LIN {X 0,Y 201.547,Z 410.206,A -85,B 0,C 180,E1 -21878.269,E2 -21878.269} C_VEL
LIN {X 0,Y 203.427,Z 397.935,A -85,B 0,C 180,E1 -21879.946,E2 -21879.946} C_VEL
LIN {X 0,Y 205.038,Z 385.054,A -85,B 0,C 180,E1 -21881.241,E2 -21881.241} C_VEL
LIN {X 0,Y 206.208,Z 372.059,A -85,B 0,C 180,E1 -21882.113,E2 -21882.113} C_VEL
LIN {X 0,Y 207.148,Z 353.067,A -85,B 0,C 180,E1 -21882.84,E2 -21882.84} C_VEL
LIN {X 0,Y 209.063,Z 305.006,A -85,B 0,C 180,E1 -21884.444,E2 -21884.444} C_VEL
LIN {X 0,Y 207.505,Z 298.752,A -85,B 0,C 180,E1 -21884.902,E2 -21884.902} C_VEL
LIN {X 0,Y 201.853,Z 283.207,A -85,B 0,C 180,E1 -21886.329,E2 -21886.329} C_VEL
LIN {X 0,Y 196.318,Z 270.427,A -85,B 0,C 180,E1 -21887.718,E2 -21887.718} C_VEL
LIN {X 0,Y 192.917,Z 263.876,A -85,B 0,C 180,E1 -21888.63,E2 -21888.63} C_VEL
LIN {X 0,Y 192.707,Z 263.031,A -85,B 0,C 180,E1 -21889.108,E2 -21889.108} C_VEL
LIN {X 0,Y 192.636,Z 262.96,A -85,B 0,C 180,E1 -21894.234,E2 -21894.234} C_VEL
LIN {X 0,Y 192.624,Z 262.95,A -85,B 0,C 180,E1 -21898.902,E2 -21898.902} C_VEL
LIN {X 0,Y 192.591,Z 262.991,A -85,B 0,C 180,E1 -21903.186,E2 -21903.186} C_VEL
LIN {X 0,Y 192.616,Z 262.98,A -85,B 0,C 180,E1 -21906.629,E2 -21906.629} C_VEL
LIN {X 0,Y 192.586,Z 262.973,A -85,B 0,C 180,E1 -21911.061,E2 -21911.061} C_VEL
LIN {X 0,Y 192.602,Z 262.994,A -85,B 0,C 180,E1 -21916.123,E2 -21916.123} C_VEL
LIN {X 0,Y 192.589,Z 262.963,A -85,B 0,C 180,E1 -21920.025,E2 -21920.025} C_VEL
LIN {X 0,Y 192.579,Z 262.983,A -85,B 0,C 180,E1 -21924.288,E2 -21924.288} C_VEL
LIN {X 0,Y 192.587,Z 262.975,A -85,B 0,C 180,E1 -21929.289,E2 -21929.289} C_VEL
LIN {X 0,Y 192.646,Z 262.94,A -85,B 0,C 180,E1 -21931.701,E2 -21931.701} C_VEL
LIN {X 0,Y 192.698,Z 262.972,A -85,B 0,C 180,E1 -21936.359,E2 -21936.359} C_VEL
LIN {X 0,Y 192.769,Z 262.951,A -85,B 0,C 180,E1 -21941.422,E2 -21941.422} C_VEL
LIN {X 0,Y 192.757,Z 262.917,A -85,B 0,C 180,E1 -21945.224,E2 -21945.224} C_VEL
LIN {X 0,Y 193.012,Z 262.934,A -85,B 0,C 180,E1 -21949.52,E2 -21949.52} C_VEL
LIN {X 0,Y 192.998,Z 262.931,A -85,B 0,C 180,E1 -21953.738,E2 -21953.738} C_VEL
LIN {X 0,Y 193.26,Z 262.855,A -85,B 0,C 180,E1 -21957.925,E2 -21957.925} C_VEL
LIN {X 0,Y 193.438,Z 262.85,A -85,B 0,C 180,E1 -21960.009,E2 -21960.009} C_VEL
LIN {X 0,Y 192.966,Z 262.949,A -85,B 0,C 180,E1 -21964.186,E2 -21964.186} C_VEL
LIN {X 0,Y 193.027,Z 262.904,A -85,B 0,C 180,E1 -21968.383,E2 -21968.383} C_VEL
LIN {X 0,Y 192.805,Z 262.941,A -85,B 0,C 180,E1 -21972.642,E2 -21972.642} C_VEL
LIN {X 0,Y 192.763,Z 262.97,A -85,B 0,C 180,E1 -21976.967,E2 -21976.967} C_VEL
LIN {X 0,Y 192.623,Z 262.954,A -85,B 0,C 180,E1 -21981.408,E2 -21981.408} C_VEL
LIN {X 0,Y 192.656,Z 262.982,A -85,B 0,C 180,E1 -21984.221,E2 -21984.221} C_VEL
LIN {X 0,Y 192.639,Z 262.965,A -85,B 0,C 180,E1 -21988.887,E2 -21988.887} C_VEL
LIN {X 0,Y 192.607,Z 262.996,A -85,B 0,C 180,E1 -21993.194,E2 -21993.194} C_VEL
LIN {X 0,Y 192.562,Z 262.985,A -85,B 0,C 180,E1 -21998.359,E2 -21998.359} C_VEL
LIN {X 0,Y 192.503,Z 262.965,A -85,B 0,C 180,E1 -22003.101,E2 -22003.101} C_VEL
LIN {X 0,Y 192.499,Z 262.962,A -85,B 0,C 180,E1 -22006.913,E2 -22006.913} C_VEL
LIN {X 0,Y 192.609,Z 263.147,A -85,B 0,C 180,E1 -22011.738,E2 -22011.738} C_VEL
LIN {X 0,Y 193.411,Z 266.363,A -85,B 0,C 180,E1 -22013.384,E2 -22013.384} C_VEL
LIN {X 0,Y 198.115,Z 277.207,A -85,B 0,C 180,E1 -22014.69,E2 -22014.69} C_VEL
LIN {X 0,Y 204.165,Z 292.827,A -85,B 0,C 180,E1 -22016.231,E2 -22016.231} C_VEL
LIN {X 0,Y 206.841,Z 301.139,A -85,B 0,C 180,E1 -22016.932,E2 -22016.932} C_VEL
LIN {X 0,Y 207.153,Z 303.933,A -85,B 0,C 180,E1 -22017.085,E2 -22017.085} C_VEL
LIN {X 0,Y 207.117,Z 309.784,A -85,B 0,C 180,E1 -22017.309,E2 -22017.309} C_VEL
LIN {X 0,Y 206.092,Z 315.639,A -85,B 0,C 180,E1 -22017.398,E2 -22017.398} C_VEL
LIN {X 0,Y 202.165,Z 331.222,A -85,B 0,C 180,E1 -22017.472,E2 -22017.472} C_VEL
LIN {X 0,Y 201.68,Z 335.194,A -85,B 0,C 180,E1 -22017.564,E2 -22017.564} C_VEL
LIN {X 0,Y 199.95,Z 375.022,A -85,B 0,C 180,E1 -22018.994,E2 -22018.994} C_VEL
LIN {X 0,Y 198.708,Z 387.932,A -85,B 0,C 180,E1 -22019.809,E2 -22019.809} C_VEL
LIN {X 0,Y 197.203,Z 399.987,A -85,B 0,C 180,E1 -22020.951,E2 -22020.951} C_VEL
LIN {X 0,Y 195.348,Z 411.355,A -85,B 0,C 180,E1 -22022.407,E2 -22022.407} C_VEL
LIN {X 0,Y 193.289,Z 421.772,A -85,B 0,C 180,E1 -22024.132,E2 -22024.132} C_VEL
LIN {X 0,Y 191.373,Z 431.488,A -85,B 0,C 180,E1 -22026.175,E2 -22026.175} C_VEL
LIN {X 0,Y 189.178,Z 441.365,A -85,B 0,C 180,E1 -22028.765,E2 -22028.765} C_VEL
LIN {X 0,Y 187.317,Z 449.442,A -85,B 0,C 180,E1 -22031.404,E2 -22031.404} C_VEL
LIN {X 0,Y 185.503,Z 457.32,A -85,B 0,C 180,E1 -22034.622,E2 -22034.622} C_VEL
LIN {X 0,Y 184.314,Z 463.61,A -85,B 0,C 180,E1 -22037.895,E2 -22037.895} C_VEL
LIN {X 0,Y 183.529,Z 468.588,A -85,B 0,C 180,E1 -22041.19,E2 -22041.19} C_VEL
LIN {X 0,Y 183.125,Z 472.408,A -85,B 0,C 180,E1 -22044.495,E2 -22044.495} C_VEL
LIN {X 0,Y 183.015,Z 475.181,A -85,B 0,C 180,E1 -22047.8,E2 -22047.8} C_VEL
LIN {X 0,Y 183.092,Z 476.483,A -85,B 0,C 180,E1 -22050.001,E2 -22050.001} C_VEL
LIN {X 0,Y 182.991,Z 477.585,A -85,B 0,C 180,E1 -22052.933,E2 -22052.933} C_VEL
LIN {X 0,Y 183.323,Z 477.96,A -85,B 0,C 180,E1 -22056.605,E2 -22056.605} C_VEL
LIN {X 0,Y 184.27,Z 476.977,A -85,B 0,C 180,E1 -22060.994,E2 -22060.994} C_VEL
LIN {X 0,Y 185.114,Z 475.917,A -85,B 0,C 180,E1 -22063.168,E2 -22063.168} C_VEL
LIN {X 0,Y 186.18,Z 474.422,A -85,B 0,C 180,E1 -22065.322,E2 -22065.322} C_VEL
LIN {X 0,Y 188.237,Z 471.426,A -85,B 0,C 180,E1 -22068.504,E2 -22068.504} C_VEL
LIN {X 0,Y 191.001,Z 467.404,A -85,B 0,C 180,E1 -22071.59,E2 -22071.59} C_VEL
LIN {X 0,Y 194.227,Z 462.258,A -85,B 0,C 180,E1 -22074.591,E2 -22074.591} C_VEL
LIN {X 0,Y 197.75,Z 455.833,A -85,B 0,C 180,E1 -22077.518,E2 -22077.518} C_VEL
LIN {X 0,Y 202.024,Z 447.849,A -85,B 0,C 180,E1 -22080.294,E2 -22080.294} C_VEL
LIN {X 0,Y 205.946,Z 439.728,A -85,B 0,C 180,E1 -22082.513,E2 -22082.513} C_VEL
LIN {X 0,Y 210.3,Z 429.83,A -85,B 0,C 180,E1 -22084.62,E2 -22084.62} C_VEL
LIN {X 0,Y 213.87,Z 420.103,A -85,B 0,C 180,E1 -22086.264,E2 -22086.264} C_VEL
LIN {X 0,Y 217.703,Z 407.824,A -85,B 0,C 180,E1 -22087.834,E2 -22087.834} C_VEL
LIN {X 0,Y 220.715,Z 395.821,A -85,B 0,C 180,E1 -22088.968,E2 -22088.968} C_VEL
LIN {X 0,Y 223.081,Z 382.949,A -85,B 0,C 180,E1 -22089.828,E2 -22089.828} C_VEL
LIN {X 0,Y 224.603,Z 369.194,A -85,B 0,C 180,E1 -22090.426,E2 -22090.426} C_VEL
LIN {X 0,Y 226.979,Z 331.617,A -85,B 0,C 180,E1 -22091.565,E2 -22091.565} C_VEL
LIN {X 0,Y 221.2,Z 318.428,A -85,B 0,C 180,E1 -22093.951,E2 -22093.951} C_VEL
LIN {X 0,Y 215.551,Z 307.564,A -85,B 0,C 180,E1 -22096.435,E2 -22096.435} C_VEL
LIN {X 0,Y 209.904,Z 297.83,A -85,B 0,C 180,E1 -22099.202,E2 -22099.202} C_VEL
LIN {X 0,Y 206.451,Z 292.45,A -85,B 0,C 180,E1 -22101.042,E2 -22101.042} C_VEL
LIN {X 0,Y 203.699,Z 288.268,A -85,B 0,C 180,E1 -22102.617,E2 -22102.617} C_VEL
LIN {X 0,Y 199.882,Z 282.7,A -85,B 0,C 180,E1 -22104.997,E2 -22104.997} C_VEL
LIN {X 0,Y 196.957,Z 278.784,A -85,B 0,C 180,E1 -22107.023,E2 -22107.023} C_VEL
LIN {X 0,Y 195.987,Z 277.356,A -85,B 0,C 180,E1 -22107.763,E2 -22107.763} C_VEL
LIN {X 0,Y 190.543,Z 270.611,A -85,B 0,C 180,E1 -22112.417,E2 -22112.417} C_VEL
LIN {X 0,Y 188.641,Z 268.893,A -85,B 0,C 180,E1 -22114.326,E2 -22114.326} C_VEL
LIN {X 0,Y 186.363,Z 266.371,A -85,B 0,C 180,E1 -22117.105,E2 -22117.105} C_VEL
LIN {X 0,Y 185.613,Z 264.245,A -85,B 0,C 180,E1 -22118.763,E2 -22118.763} C_VEL
LIN {X 0,Y 185.542,Z 263.873,A -85,B 0,C 180,E1 -22120.059,E2 -22120.059} C_VEL
LIN {X 0,Y 185.663,Z 263.859,A -85,B 0,C 180,E1 -22122.363,E2 -22122.363} C_VEL
LIN {X 0,Y 185.726,Z 263.851,A -85,B 0,C 180,E1 -22126.868,E2 -22126.868} C_VEL
LIN {X 0,Y 185.984,Z 263.817,A -85,B 0,C 180,E1 -22131.297,E2 -22131.297} C_VEL
LIN {X 0,Y 186.185,Z 263.778,A -85,B 0,C 180,E1 -22137.827,E2 -22137.827} C_VEL
LIN {X 0,Y 186.399,Z 263.758,A -85,B 0,C 180,E1 -22139.99,E2 -22139.99} C_VEL
LIN {X 0,Y 185.946,Z 264.019,A -85,B 0,C 180,E1 -22144.19,E2 -22144.19} C_VEL
LIN {X 0,Y 186.707,Z 266.344,A -85,B 0,C 180,E1 -22145.525,E2 -22145.525} C_VEL
LIN {X 0,Y 188.785,Z 268.646,A -85,B 0,C 180,E1 -22148.015,E2 -22148.015} C_VEL
LIN {X 0,Y 190.993,Z 269.918,A -85,B 0,C 180,E1 -22150.115,E2 -22150.115} C_VEL
LIN {X 0,Y 192.307,Z 272.671,A -85,B 0,C 180,E1 -22151.452,E2 -22151.452} C_VEL
LIN {X 0,Y 194.404,Z 274.827,A -85,B 0,C 180,E1 -22153.185,E2 -22153.185} C_VEL
LIN {X 0,Y 195.644,Z 275.781,A -85,B 0,C 180,E1 -22154.107,E2 -22154.107} C_VEL
LIN {X 0,Y 197.722,Z 279.021,A -85,B 0,C 180,E1 -22155.699,E2 -22155.699} C_VEL
LIN {X 0,Y 199.843,Z 281.118,A -85,B 0,C 180,E1 -22157.093,E2 -22157.093} C_VEL
LIN {X 0,Y 202.443,Z 284.707,A -85,B 0,C 180,E1 -22158.738,E2 -22158.738} C_VEL
LIN {X 0,Y 204.939,Z 288.002,A -85,B 0,C 180,E1 -22160.192,E2 -22160.192} C_VEL
LIN {X 0,Y 208.483,Z 293.32,A -85,B 0,C 180,E1 -22162.146,E2 -22162.146} C_VEL
LIN {X 0,Y 211.835,Z 298.487,A -85,B 0,C 180,E1 -22163.854,E2 -22163.854} C_VEL
LIN {X 0,Y 218.039,Z 309.192,A -85,B 0,C 180,E1 -22166.762,E2 -22166.762} C_VEL
LIN {X 0,Y 223.429,Z 319.688,A -85,B 0,C 180,E1 -22169.04,E2 -22169.04} C_VEL
LIN {X 0,Y 227.273,Z 328.108,A -85,B 0,C 180,E1 -22170.584,E2 -22170.584} C_VEL
LIN {X 0,Y 224.341,Z 370.593,A -85,B 0,C 180,E1 -22171.882,E2 -22171.882} C_VEL
LIN {X 0,Y 222.438,Z 383.985,A -85,B 0,C 180,E1 -22172.584,E2 -22172.584} C_VEL
LIN {X 0,Y 220.078,Z 395.902,A -85,B 0,C 180,E1 -22173.532,E2 -22173.532} C_VEL
LIN {X 0,Y 217.013,Z 407.276,A -85,B 0,C 180,E1 -22174.737,E2 -22174.737} C_VEL
LIN {X 0,Y 213.334,Z 418.666,A -85,B 0,C 180,E1 -22176.357,E2 -22176.357} C_VEL
LIN {X 0,Y 209.3,Z 429.173,A -85,B 0,C 180,E1 -22178.288,E2 -22178.288} C_VEL
LIN {X 0,Y 205.394,Z 438.08,A -85,B 0,C 180,E1 -22180.393,E2 -22180.393} C_VEL
LIN {X 0,Y 201.244,Z 446.261,A -85,B 0,C 180,E1 -22182.829,E2 -22182.829} C_VEL
LIN {X 0,Y 197.654,Z 452.831,A -85,B 0,C 180,E1 -22185.312,E2 -22185.312} C_VEL
LIN {X 0,Y 194.299,Z 458.472,A -85,B 0,C 180,E1 -22187.997,E2 -22187.997} C_VEL
LIN {X 0,Y 190.893,Z 463.723,A -85,B 0,C 180,E1 -22191.253,E2 -22191.253} C_VEL
LIN {X 0,Y 188.11,Z 467.703,A -85,B 0,C 180,E1 -22194.614,E2 -22194.614} C_VEL
LIN {X 0,Y 185.932,Z 470.52,A -85,B 0,C 180,E1 -22198.049,E2 -22198.049} C_VEL
LIN {X 0,Y 184.527,Z 472.119,A -85,B 0,C 180,E1 -22201.137,E2 -22201.137} C_VEL
LIN {X 0,Y 183.33,Z 472.982,A -85,B 0,C 180,E1 -22205.058,E2 -22205.058} C_VEL
LIN {X 0,Y 182.955,Z 472.916,A -85,B 0,C 180,E1 -22207.409,E2 -22207.409} C_VEL
LIN {X 0,Y 182.676,Z 472.397,A -85,B 0,C 180,E1 -22209.741,E2 -22209.741} C_VEL
LIN {X 0,Y 182.641,Z 470.206,A -85,B 0,C 180,E1 -22214.108,E2 -22214.108} C_VEL
LIN {X 0,Y 183.078,Z 467.071,A -85,B 0,C 180,E1 -22217.81,E2 -22217.81} C_VEL
LIN {X 0,Y 183.707,Z 463.045,A -85,B 0,C 180,E1 -22221.197,E2 -22221.197} C_VEL
LIN {X 0,Y 184.875,Z 456.83,A -85,B 0,C 180,E1 -22225.093,E2 -22225.093} C_VEL
LIN {X 0,Y 186.293,Z 450.023,A -85,B 0,C 180,E1 -22228.378,E2 -22228.378} C_VEL
LIN {X 0,Y 188.209,Z 441.565,A -85,B 0,C 180,E1 -22231.604,E2 -22231.604} C_VEL
LIN {X 0,Y 190.25,Z 432.604,A -85,B 0,C 180,E1 -22234.296,E2 -22234.296} C_VEL
LIN {X 0,Y 192.563,Z 422.034,A -85,B 0,C 180,E1 -22236.811,E2 -22236.811} C_VEL
LIN {X 0,Y 194.711,Z 411.29,A -85,B 0,C 180,E1 -22238.823,E2 -22238.823} C_VEL
LIN {X 0,Y 196.701,Z 399.301,A -85,B 0,C 180,E1 -22240.55,E2 -22240.55} C_VEL
LIN {X 0,Y 198.347,Z 386.829,A -85,B 0,C 180,E1 -22241.885,E2 -22241.885} C_VEL
LIN {X 0,Y 199.618,Z 373.948,A -85,B 0,C 180,E1 -22242.84,E2 -22242.84} C_VEL
LIN {X 0,Y 200.492,Z 358.681,A -85,B 0,C 180,E1 -22243.492,E2 -22243.492} C_VEL
LIN {X 0,Y 202.709,Z 306.126,A -85,B 0,C 180,E1 -22245.287,E2 -22245.287} C_VEL
LIN {X 0,Y 201.167,Z 300.454,A -85,B 0,C 180,E1 -22245.736,E2 -22245.736} C_VEL
LIN {X 0,Y 195.349,Z 284.469,A -85,B 0,C 180,E1 -22247.284,E2 -22247.284} C_VEL
LIN {X 0,Y 190.394,Z 273.241,A -85,B 0,C 180,E1 -22248.593,E2 -22248.593} C_VEL
LIN {X 0,Y 186.774,Z 266.912,A -85,B 0,C 180,E1 -22249.52,E2 -22249.52} C_VEL
LIN {X 0,Y 185.732,Z 264.595,A -85,B 0,C 180,E1 -22249.91,E2 -22249.91} C_VEL
LIN {X 0,Y 185.593,Z 263.913,A -85,B 0,C 180,E1 -22250.359,E2 -22250.359} C_VEL
LIN {X 0,Y 185.581,Z 263.829,A -85,B 0,C 180,E1 -22254.678,E2 -22254.678} C_VEL
LIN {X 0,Y 185.548,Z 263.839,A -85,B 0,C 180,E1 -22259.498,E2 -22259.498} C_VEL
LIN {X 0,Y 185.516,Z 263.858,A -85,B 0,C 180,E1 -22264.627,E2 -22264.627} C_VEL
LIN {X 0,Y 185.566,Z 263.865,A -85,B 0,C 180,E1 -22267.332,E2 -22267.332} C_VEL
LIN {X 0,Y 185.564,Z 263.85,A -85,B 0,C 180,E1 -22270.776,E2 -22270.776} C_VEL
LIN {X 0,Y 185.56,Z 263.87,A -85,B 0,C 180,E1 -22276.022,E2 -22276.022} C_VEL
LIN {X 0,Y 185.541,Z 263.841,A -85,B 0,C 180,E1 -22279.929,E2 -22279.929} C_VEL
LIN {X 0,Y 185.551,Z 263.837,A -85,B 0,C 180,E1 -22282.712,E2 -22282.712} C_VEL
LIN {X 0,Y 185.524,Z 263.869,A -85,B 0,C 180,E1 -22287.984,E2 -22287.984} C_VEL
LIN {X 0,Y 185.562,Z 263.831,A -85,B 0,C 180,E1 -22290.585,E2 -22290.585} C_VEL
LIN {X 0,Y 185.589,Z 263.845,A -85,B 0,C 180,E1 -22295.395,E2 -22295.395} C_VEL
LIN {X 0,Y 185.698,Z 263.837,A -85,B 0,C 180,E1 -22301.11,E2 -22301.11} C_VEL
LIN {X 0,Y 185.734,Z 263.806,A -85,B 0,C 180,E1 -22306.888,E2 -22306.888} C_VEL
LIN {X 0,Y 186.022,Z 263.814,A -85,B 0,C 180,E1 -22311.318,E2 -22311.318} C_VEL
LIN {X 0,Y 186.204,Z 263.732,A -85,B 0,C 180,E1 -22317.847,E2 -22317.847} C_VEL
LIN {X 0,Y 186.402,Z 263.725,A -85,B 0,C 180,E1 -22320.01,E2 -22320.01} C_VEL
LIN {X 0,Y 185.912,Z 263.827,A -85,B 0,C 180,E1 -22324.346,E2 -22324.346} C_VEL
LIN {X 0,Y 185.976,Z 263.777,A -85,B 0,C 180,E1 -22328.704,E2 -22328.704} C_VEL
LIN {X 0,Y 185.733,Z 263.827,A -85,B 0,C 180,E1 -22333.132,E2 -22333.132} C_VEL
LIN {X 0,Y 185.696,Z 263.845,A -85,B 0,C 180,E1 -22337.634,E2 -22337.634} C_VEL
LIN {X 0,Y 185.586,Z 263.836,A -85,B 0,C 180,E1 -22342.262,E2 -22342.262} C_VEL
LIN {X 0,Y 185.564,Z 263.867,A -85,B 0,C 180,E1 -22347.041,E2 -22347.041} C_VEL
LIN {X 0,Y 185.545,Z 263.862,A -85,B 0,C 180,E1 -22352.035,E2 -22352.035} C_VEL
LIN {X 0,Y 185.516,Z 263.858,A -85,B 0,C 180,E1 -22357.321,E2 -22357.321} C_VEL
LIN {X 0,Y 185.483,Z 263.879,A -85,B 0,C 180,E1 -22360.731,E2 -22360.731} C_VEL
LIN {X 0,Y 185.47,Z 263.828,A -85,B 0,C 180,E1 -22366.063,E2 -22366.063} C_VEL
LIN {X 0,Y 185.547,Z 264.033,A -85,B 0,C 180,E1 -22370.912,E2 -22370.912} C_VEL
LIN {X 0,Y 186.135,Z 266.282,A -85,B 0,C 180,E1 -22372.085,E2 -22372.085} C_VEL
LIN {X 0,Y 191.64,Z 278.578,A -85,B 0,C 180,E1 -22373.688,E2 -22373.688} C_VEL
LIN {X 0,Y 198.012,Z 295.006,A -85,B 0,C 180,E1 -22375.408,E2 -22375.408} C_VEL
LIN {X 0,Y 200.584,Z 302.839,A -85,B 0,C 180,E1 -22376.112,E2 -22376.112} C_VEL
LIN {X 0,Y 202.351,Z 318.702,A -85,B 0,C 180,E1 -22376.999,E2 -22376.999} C_VEL
LIN {X 0,Y 201.68,Z 335.194,A -85,B 0,C 180,E1 -22377.564,E2 -22377.564} C_VEL
LIN {X 0,Y 200.741,Z 341.026,A -85,B 0,C 180,E1 -22377.667,E2 -22377.667} C_VEL
LIN {X 0,Y 194.803,Z 359.947,A -85,B 0,C 180,E1 -22377.6,E2 -22377.6} C_VEL
LIN {X 0,Y 193.993,Z 365.777,A -85,B 0,C 180,E1 -22377.726,E2 -22377.726} C_VEL
LIN {X 0,Y 193.162,Z 378.83,A -85,B 0,C 180,E1 -22378.313,E2 -22378.313} C_VEL
LIN {X 0,Y 191.813,Z 391.743,A -85,B 0,C 180,E1 -22379.293,E2 -22379.293} C_VEL
LIN {X 0,Y 190.025,Z 404.235,A -85,B 0,C 180,E1 -22380.657,E2 -22380.657} C_VEL
LIN {X 0,Y 187.77,Z 416.195,A -85,B 0,C 180,E1 -22382.408,E2 -22382.408} C_VEL
LIN {X 0,Y 185.456,Z 426.9,A -85,B 0,C 180,E1 -22384.466,E2 -22384.466} C_VEL
LIN {X 0,Y 183.49,Z 436.16,A -85,B 0,C 180,E1 -22386.721,E2 -22386.721} C_VEL
LIN {X 0,Y 182.141,Z 442.349,A -85,B 0,C 180,E1 -22388.518,E2 -22388.518} C_VEL
LIN {X 0,Y 180.235,Z 450.179,A -85,B 0,C 180,E1 -22391.235,E2 -22391.235} C_VEL
LIN {X 0,Y 178.374,Z 457.858,A -85,B 0,C 180,E1 -22394.577,E2 -22394.577} C_VEL
LIN {X 0,Y 176.996,Z 464.942,A -85,B 0,C 180,E1 -22398.549,E2 -22398.549} C_VEL
LIN {X 0,Y 176.292,Z 469.612,A -85,B 0,C 180,E1 -22401.98,E2 -22401.98} C_VEL
LIN {X 0,Y 175.966,Z 473.144,A -85,B 0,C 180,E1 -22405.419,E2 -22405.419} C_VEL
LIN {X 0,Y 175.932,Z 474.924,A -85,B 0,C 180,E1 -22407.711,E2 -22407.711} C_VEL
LIN {X 0,Y 176.004,Z 476.261,A -85,B 0,C 180,E1 -22410.001,E2 -22410.001} C_VEL
LIN {X 0,Y 175.917,Z 477.331,A -85,B 0,C 180,E1 -22412.689,E2 -22412.689} C_VEL
LIN {X 0,Y 176.263,Z 477.879,A -85,B 0,C 180,E1 -22416.871,E2 -22416.871} C_VEL
LIN {X 0,Y 177.29,Z 476.972,A -85,B 0,C 180,E1 -22421.433,E2 -22421.433} C_VEL
LIN {X 0,Y 179.31,Z 474.538,A -85,B 0,C 180,E1 -22425.925,E2 -22425.925} C_VEL
LIN {X 0,Y 181.514,Z 471.61,A -85,B 0,C 180,E1 -22429.215,E2 -22429.215} C_VEL
LIN {X 0,Y 184.435,Z 467.667,A -85,B 0,C 180,E1 -22432.4,E2 -22432.4} C_VEL
LIN {X 0,Y 187.781,Z 462.625,A -85,B 0,C 180,E1 -22435.494,E2 -22435.494} C_VEL
LIN {X 0,Y 191.513,Z 456.323,A -85,B 0,C 180,E1 -22438.494,E2 -22438.494} C_VEL
LIN {X 0,Y 195.968,Z 448.461,A -85,B 0,C 180,E1 -22441.334,E2 -22441.334} C_VEL
LIN {X 0,Y 200.045,Z 440.479,A -85,B 0,C 180,E1 -22443.596,E2 -22443.596} C_VEL
LIN {X 0,Y 204.555,Z 430.753,A -85,B 0,C 180,E1 -22445.738,E2 -22445.738} C_VEL
LIN {X 0,Y 208.233,Z 421.265,A -85,B 0,C 180,E1 -22447.41,E2 -22447.41} C_VEL
LIN {X 0,Y 211.71,Z 411.072,A -85,B 0,C 180,E1 -22448.799,E2 -22448.799} C_VEL
LIN {X 0,Y 215.053,Z 398.966,A -85,B 0,C 180,E1 -22450.046,E2 -22450.046} C_VEL
LIN {X 0,Y 217.849,Z 385.297,A -85,B 0,C 180,E1 -22451.051,E2 -22451.051} C_VEL
LIN {X 0,Y 219.562,Z 372.451,A -85,B 0,C 180,E1 -22451.671,E2 -22451.671} C_VEL
LIN {X 0,Y 222.189,Z 334.267,A -85,B 0,C 180,E1 -22452.837,E2 -22452.837} C_VEL
LIN {X 0,Y 216.303,Z 320.689,A -85,B 0,C 180,E1 -22455.439,E2 -22455.439} C_VEL
LIN {X 0,Y 209.977,Z 308.591,A -85,B 0,C 180,E1 -22458.504,E2 -22458.504} C_VEL
LIN {X 0,Y 204.622,Z 299.506,A -85,B 0,C 180,E1 -22461.399,E2 -22461.399} C_VEL
LIN {X 0,Y 200.725,Z 293.589,A -85,B 0,C 180,E1 -22463.724,E2 -22463.724} C_VEL
LIN {X 0,Y 197.536,Z 288.77,A -85,B 0,C 180,E1 -22465.833,E2 -22465.833} C_VEL
LIN {X 0,Y 194.597,Z 284.573,A -85,B 0,C 180,E1 -22468.014,E2 -22468.014} C_VEL
LIN {X 0,Y 188.941,Z 277.217,A -85,B 0,C 180,E1 -22473.049,E2 -22473.049} C_VEL
LIN {X 0,Y 186.851,Z 275.38,A -85,B 0,C 180,E1 -22475.254,E2 -22475.254} C_VEL
LIN {X 0,Y 184.672,Z 272.412,A -85,B 0,C 180,E1 -22478.21,E2 -22478.21} C_VEL
LIN {X 0,Y 184.048,Z 270.965,A -85,B 0,C 180,E1 -22479.306,E2 -22479.306} C_VEL
LIN {X 0,Y 180.36,Z 268.256,A -85,B 0,C 180,E1 -22489.817,E2 -22489.817} C_VEL
LIN {X 0,Y 180.513,Z 268.417,A -85,B 0,C 180,E1 -22493.844,E2 -22493.844} C_VEL
LIN {X 0,Y 182.967,Z 270.052,A -85,B 0,C 180,E1 -22501.089,E2 -22501.089} C_VEL
LIN {X 0,Y 184.536,Z 270.998,A -85,B 0,C 180,E1 -22503.606,E2 -22503.606} C_VEL
LIN {X 0,Y 185.662,Z 273.583,A -85,B 0,C 180,E1 -22505.42,E2 -22505.42} C_VEL
LIN {X 0,Y 187.893,Z 275.775,A -85,B 0,C 180,E1 -22508.053,E2 -22508.053} C_VEL
LIN {X 0,Y 189.338,Z 276.801,A -85,B 0,C 180,E1 -22509.482,E2 -22509.482} C_VEL
LIN {X 0,Y 191.025,Z 279.801,A -85,B 0,C 180,E1 -22511.194,E2 -22511.194} C_VEL
LIN {X 0,Y 193.787,Z 282.496,A -85,B 0,C 180,E1 -22513.48,E2 -22513.48} C_VEL
LIN {X 0,Y 196.205,Z 285.965,A -85,B 0,C 180,E1 -22515.368,E2 -22515.368} C_VEL
LIN {X 0,Y 197.701,Z 287.52,A -85,B 0,C 180,E1 -22516.396,E2 -22516.396} C_VEL
LIN {X 0,Y 200.408,Z 291.179,A -85,B 0,C 180,E1 -22518.166,E2 -22518.166} C_VEL
LIN {X 0,Y 204.913,Z 297.764,A -85,B 0,C 180,E1 -22520.851,E2 -22520.851} C_VEL
LIN {X 0,Y 209.878,Z 305.794,A -85,B 0,C 180,E1 -22523.517,E2 -22523.517} C_VEL
LIN {X 0,Y 215.869,Z 316.667,A -85,B 0,C 180,E1 -22526.426,E2 -22526.426} C_VEL
LIN {X 0,Y 221.933,Z 329.453,A -85,B 0,C 180,E1 -22529.076,E2 -22529.076} C_VEL
LIN {X 0,Y 222.44,Z 330.733,A -85,B 0,C 180,E1 -22529.295,E2 -22529.295} C_VEL
LIN {X 0,Y 219.613,Z 370.172,A -85,B 0,C 180,E1 -22530.504,E2 -22530.504} C_VEL
LIN {X 0,Y 217.582,Z 384.057,A -85,B 0,C 180,E1 -22531.228,E2 -22531.228} C_VEL
LIN {X 0,Y 214.998,Z 396.565,A -85,B 0,C 180,E1 -22532.24,E2 -22532.24} C_VEL
LIN {X 0,Y 211.734,Z 408.106,A -85,B 0,C 180,E1 -22533.491,E2 -22533.491} C_VEL
LIN {X 0,Y 207.659,Z 420.058,A -85,B 0,C 180,E1 -22535.241,E2 -22535.241} C_VEL
LIN {X 0,Y 203.714,Z 429.746,A -85,B 0,C 180,E1 -22537.079,E2 -22537.079} C_VEL
LIN {X 0,Y 199.359,Z 439.105,A -85,B 0,C 180,E1 -22539.373,E2 -22539.373} C_VEL
LIN {X 0,Y 194.521,Z 448.11,A -85,B 0,C 180,E1 -22542.212,E2 -22542.212} C_VEL
LIN {X 0,Y 190.053,Z 455.645,A -85,B 0,C 180,E1 -22545.363,E2 -22545.363} C_VEL
LIN {X 0,Y 186.267,Z 461.329,A -85,B 0,C 180,E1 -22548.497,E2 -22548.497} C_VEL
LIN {X 0,Y 182.857,Z 466.101,A -85,B 0,C 180,E1 -22552.051,E2 -22552.051} C_VEL
LIN {X 0,Y 180.829,Z 468.743,A -85,B 0,C 180,E1 -22554.683,E2 -22554.683} C_VEL
LIN {X 0,Y 178.224,Z 471.685,A -85,B 0,C 180,E1 -22559.16,E2 -22559.16} C_VEL
LIN {X 0,Y 177.214,Z 472.614,A -85,B 0,C 180,E1 -22561.581,E2 -22561.581} C_VEL
LIN {X 0,Y 176.471,Z 473.052,A -85,B 0,C 180,E1 -22564.018,E2 -22564.018} C_VEL
LIN {X 0,Y 175.953,Z 473.037,A -85,B 0,C 180,E1 -22566.701,E2 -22566.701} C_VEL
LIN {X 0,Y 175.649,Z 472.642,A -85,B 0,C 180,E1 -22568.893,E2 -22568.893} C_VEL
LIN {X 0,Y 175.484,Z 471.767,A -85,B 0,C 180,E1 -22571.313,E2 -22571.313} C_VEL
LIN {X 0,Y 175.54,Z 470.348,A -85,B 0,C 180,E1 -22573.873,E2 -22573.873} C_VEL
LIN {X 0,Y 175.883,Z 467.628,A -85,B 0,C 180,E1 -22577.304,E2 -22577.304} C_VEL
LIN {X 0,Y 176.518,Z 463.748,A -85,B 0,C 180,E1 -22580.835,E2 -22580.835} C_VEL
LIN {X 0,Y 177.487,Z 458.706,A -85,B 0,C 180,E1 -22584.318,E2 -22584.318} C_VEL
LIN {X 0,Y 178.846,Z 452.362,A -85,B 0,C 180,E1 -22587.747,E2 -22587.747} C_VEL
LIN {X 0,Y 180.658,Z 444.423,A -85,B 0,C 180,E1 -22591.114,E2 -22591.114} C_VEL
LIN {X 0,Y 182.588,Z 436.291,A -85,B 0,C 180,E1 -22593.862,E2 -22593.862} C_VEL
LIN {X 0,Y 184.952,Z 426.338,A -85,B 0,C 180,E1 -22596.545,E2 -22596.545} C_VEL
LIN {X 0,Y 187.054,Z 416.574,A -85,B 0,C 180,E1 -22598.643,E2 -22598.643} C_VEL
LIN {X 0,Y 189.07,Z 406.042,A -85,B 0,C 180,E1 -22600.44,E2 -22600.44} C_VEL
LIN {X 0,Y 191.029,Z 393.385,A -85,B 0,C 180,E1 -22602.077,E2 -22602.077} C_VEL
LIN {X 0,Y 192.613,Z 380.019,A -85,B 0,C 180,E1 -22603.316,E2 -22603.316} C_VEL
LIN {X 0,Y 193.664,Z 367.623,A -85,B 0,C 180,E1 -22604.044,E2 -22604.044} C_VEL
LIN {X 0,Y 196.392,Z 307.179,A -85,B 0,C 180,E1 -22606.174,E2 -22606.174} C_VEL
LIN {X 0,Y 192.279,Z 294.653,A -85,B 0,C 180,E1 -22607.35,E2 -22607.35} C_VEL
LIN {X 0,Y 186.156,Z 279.354,A -85,B 0,C 180,E1 -22609.074,E2 -22609.074} C_VEL
LIN {X 0,Y 181.645,Z 271.163,A -85,B 0,C 180,E1 -22610.296,E2 -22610.296} C_VEL
LIN {X 0,Y 178.723,Z 265.614,A -85,B 0,C 180,E1 -22611.201,E2 -22611.201} C_VEL
LIN {X 0,Y 178.57,Z 264.791,A -85,B 0,C 180,E1 -22611.703,E2 -22611.703} C_VEL
LIN {X 0,Y 178.485,Z 264.7,A -85,B 0,C 180,E1 -22615.666,E2 -22615.666} C_VEL
LIN {X 0,Y 178.476,Z 264.745,A -85,B 0,C 180,E1 -22620.79,E2 -22620.79} C_VEL
LIN {X 0,Y 178.485,Z 264.736,A -85,B 0,C 180,E1 -22624.241,E2 -22624.241} C_VEL
LIN {X 0,Y 178.473,Z 264.754,A -85,B 0,C 180,E1 -22629.053,E2 -22629.053} C_VEL
LIN {X 0,Y 178.489,Z 264.722,A -85,B 0,C 180,E1 -22632.018,E2 -22632.018} C_VEL
LIN {X 0,Y 178.502,Z 264.742,A -85,B 0,C 180,E1 -22635.128,E2 -22635.128} C_VEL
LIN {X 0,Y 178.493,Z 264.739,A -85,B 0,C 180,E1 -22638.425,E2 -22638.425} C_VEL
LIN {X 0,Y 178.445,Z 264.735,A -85,B 0,C 180,E1 -22643.803,E2 -22643.803} C_VEL
LIN {X 0,Y 178.469,Z 264.755,A -85,B 0,C 180,E1 -22646.557,E2 -22646.557} C_VEL
LIN {X 0,Y 178.503,Z 264.716,A -85,B 0,C 180,E1 -22650.016,E2 -22650.016} C_VEL
LIN {X 0,Y 178.518,Z 264.718,A -85,B 0,C 180,E1 -22654.885,E2 -22654.885} C_VEL
LIN {X 0,Y 178.642,Z 264.718,A -85,B 0,C 180,E1 -22660.765,E2 -22660.765} C_VEL
LIN {X 0,Y 178.658,Z 264.679,A -85,B 0,C 180,E1 -22666.359,E2 -22666.359} C_VEL
LIN {X 0,Y 178.971,Z 264.69,A -85,B 0,C 180,E1 -22670.973,E2 -22670.973} C_VEL
LIN {X 0,Y 179.15,Z 264.61,A -85,B 0,C 180,E1 -22677.762,E2 -22677.762} C_VEL
LIN {X 0,Y 179.365,Z 264.6,A -85,B 0,C 180,E1 -22680.01,E2 -22680.01} C_VEL
LIN {X 0,Y 178.86,Z 264.705,A -85,B 0,C 180,E1 -22684.517,E2 -22684.517} C_VEL
LIN {X 0,Y 178.907,Z 264.653,A -85,B 0,C 180,E1 -22689.05,E2 -22689.05} C_VEL
LIN {X 0,Y 178.661,Z 264.715,A -85,B 0,C 180,E1 -22693.662,E2 -22693.662} C_VEL
LIN {X 0,Y 178.628,Z 264.705,A -85,B 0,C 180,E1 -22699.223,E2 -22699.223} C_VEL
LIN {X 0,Y 178.529,Z 264.748,A -85,B 0,C 180,E1 -22705.122,E2 -22705.122} C_VEL
LIN {X 0,Y 178.475,Z 264.729,A -85,B 0,C 180,E1 -22710.802,E2 -22710.802} C_VEL
LIN {X 0,Y 178.495,Z 264.755,A -85,B 0,C 180,E1 -22714.226,E2 -22714.226} C_VEL
LIN {X 0,Y 178.407,Z 264.755,A -85,B 0,C 180,E1 -22719.082,E2 -22719.082} C_VEL
LIN {X 0,Y 178.412,Z 264.735,A -85,B 0,C 180,E1 -22722.052,E2 -22722.052} C_VEL
LIN {X 0,Y 178.407,Z 264.704,A -85,B 0,C 180,E1 -22725.172,E2 -22725.172} C_VEL
LIN {X 0,Y 178.468,Z 264.928,A -85,B 0,C 180,E1 -22730.014,E2 -22730.014} C_VEL
LIN {X 0,Y 178.853,Z 266.384,A -85,B 0,C 180,E1 -22730.692,E2 -22730.692} C_VEL
LIN {X 0,Y 184.54,Z 278.407,A -85,B 0,C 180,E1 -22732.421,E2 -22732.421} C_VEL
LIN {X 0,Y 191.911,Z 297.171,A -85,B 0,C 180,E1 -22734.533,E2 -22734.533} C_VEL
LIN {X 0,Y 194.453,Z 305.297,A -85,B 0,C 180,E1 -22735.284,E2 -22735.284} C_VEL
LIN {X 0,Y 196,Z 320.651,A -85,B 0,C 180,E1 -22736.159,E2 -22736.159} C_VEL
LIN {X 0,Y 193.993,Z 365.777,A -85,B 0,C 180,E1 -22737.726,E2 -22737.726} C_VEL
LIN {X 0,Y 193.188,Z 369.683,A -85,B 0,C 180,E1 -22737.783,E2 -22737.783} C_VEL
LIN {X 0,Y 190.164,Z 375.737,A -85,B 0,C 180,E1 -22737.681,E2 -22737.681} C_VEL
LIN {X 0,Y 187.022,Z 381.726,A -85,B 0,C 180,E1 -22737.665,E2 -22737.665} C_VEL
LIN {X 0,Y 186.031,Z 385.527,A -85,B 0,C 180,E1 -22737.868,E2 -22737.868} C_VEL
LIN {X 0,Y 184.314,Z 399.04,A -85,B 0,C 180,E1 -22739.179,E2 -22739.179} C_VEL
LIN {X 0,Y 182.142,Z 411.433,A -85,B 0,C 180,E1 -22740.848,E2 -22740.848} C_VEL
LIN {X 0,Y 180.192,Z 420.474,A -85,B 0,C 180,E1 -22742.41,E2 -22742.41} C_VEL
LIN {X 0,Y 178.091,Z 430.399,A -85,B 0,C 180,E1 -22744.587,E2 -22744.587} C_VEL
LIN {X 0,Y 175.518,Z 440.877,A -85,B 0,C 180,E1 -22747.489,E2 -22747.489} C_VEL
LIN {X 0,Y 173.449,Z 449.387,A -85,B 0,C 180,E1 -22750.472,E2 -22750.472} C_VEL
LIN {X 0,Y 171.484,Z 457.231,A -85,B 0,C 180,E1 -22753.941,E2 -22753.941} C_VEL
LIN {X 0,Y 170.022,Z 464.419,A -85,B 0,C 180,E1 -22758.073,E2 -22758.073} C_VEL
LIN {X 0,Y 169.236,Z 469.179,A -85,B 0,C 180,E1 -22761.643,E2 -22761.643} C_VEL
LIN {X 0,Y 168.887,Z 472.796,A -85,B 0,C 180,E1 -22765.227,E2 -22765.227} C_VEL
LIN {X 0,Y 168.842,Z 474.649,A -85,B 0,C 180,E1 -22767.615,E2 -22767.615} C_VEL
LIN {X 0,Y 168.904,Z 476.029,A -85,B 0,C 180,E1 -22770.001,E2 -22770.001} C_VEL
LIN {X 0,Y 168.842,Z 477,A -85,B 0,C 180,E1 -22772.386,E2 -22772.386} C_VEL
LIN {X 0,Y 169.198,Z 477.789,A -85,B 0,C 180,E1 -22777.159,E2 -22777.159} C_VEL
LIN {X 0,Y 170.329,Z 476.97,A -85,B 0,C 180,E1 -22781.907,E2 -22781.907} C_VEL
LIN {X 0,Y 172.463,Z 474.629,A -85,B 0,C 180,E1 -22786.575,E2 -22786.575} C_VEL
LIN {X 0,Y 174.823,Z 471.77,A -85,B 0,C 180,E1 -22789.981,E2 -22789.981} C_VEL
LIN {X 0,Y 177.892,Z 467.912,A -85,B 0,C 180,E1 -22793.271,E2 -22793.271} C_VEL
LIN {X 0,Y 181.389,Z 462.964,A -85,B 0,C 180,E1 -22796.461,E2 -22796.461} C_VEL
LIN {X 0,Y 185.313,Z 456.783,A -85,B 0,C 180,E1 -22799.54,E2 -22799.54} C_VEL
LIN {X 0,Y 189.985,Z 449.072,A -85,B 0,C 180,E1 -22802.439,E2 -22802.439} C_VEL
LIN {X 0,Y 195.16,Z 439.461,A -85,B 0,C 180,E1 -22805.183,E2 -22805.183} C_VEL
LIN {X 0,Y 199.834,Z 429.553,A -85,B 0,C 180,E1 -22807.35,E2 -22807.35} C_VEL
LIN {X 0,Y 203.721,Z 419.8,A -85,B 0,C 180,E1 -22809.021,E2 -22809.021} C_VEL
LIN {X 0,Y 207.875,Z 407.483,A -85,B 0,C 180,E1 -22810.604,E2 -22810.604} C_VEL
LIN {X 0,Y 211.088,Z 395.445,A -85,B 0,C 180,E1 -22811.751,E2 -22811.751} C_VEL
LIN {X 0,Y 213.649,Z 382.263,A -85,B 0,C 180,E1 -22812.627,E2 -22812.627} C_VEL
LIN {X 0,Y 215.24,Z 368.781,A -85,B 0,C 180,E1 -22813.209,E2 -22813.209} C_VEL
LIN {X 0,Y 217.45,Z 336.717,A -85,B 0,C 180,E1 -22814.196,E2 -22814.196} C_VEL
LIN {X 0,Y 212.428,Z 324.981,A -85,B 0,C 180,E1 -22816.581,E2 -22816.581} C_VEL
LIN {X 0,Y 206.853,Z 313.949,A -85,B 0,C 180,E1 -22819.458,E2 -22819.458} C_VEL
LIN {X 0,Y 201.859,Z 305.199,A -85,B 0,C 180,E1 -22822.31,E2 -22822.31} C_VEL
LIN {X 0,Y 197.809,Z 298.911,A -85,B 0,C 180,E1 -22824.871,E2 -22824.871} C_VEL
LIN {X 0,Y 195.286,Z 294.895,A -85,B 0,C 180,E1 -22826.666,E2 -22826.666} C_VEL
LIN {X 0,Y 191.837,Z 289.888,A -85,B 0,C 180,E1 -22829.42,E2 -22829.42} C_VEL
LIN {X 0,Y 187.14,Z 283.541,A -85,B 0,C 180,E1 -22833.934,E2 -22833.934} C_VEL
LIN {X 0,Y 184.037,Z 280.403,A -85,B 0,C 180,E1 -22837.688,E2 -22837.688} C_VEL
LIN {X 0,Y 182.842,Z 277.857,A -85,B 0,C 180,E1 -22839.751,E2 -22839.751} C_VEL
LIN {X 0,Y 179.427,Z 275.179,A -85,B 0,C 180,E1 -22850.976,E2 -22850.976} C_VEL
LIN {X 0,Y 180.804,Z 276.299,A -85,B 0,C 180,E1 -22858.319,E2 -22858.319} C_VEL
LIN {X 0,Y 183.182,Z 277.793,A -85,B 0,C 180,E1 -22862.966,E2 -22862.966} C_VEL
LIN {X 0,Y 184.492,Z 280.586,A -85,B 0,C 180,E1 -22865.129,E2 -22865.129} C_VEL
LIN {X 0,Y 186.942,Z 282.857,A -85,B 0,C 180,E1 -22868.026,E2 -22868.026} C_VEL
LIN {X 0,Y 187.82,Z 283.748,A -85,B 0,C 180,E1 -22868.947,E2 -22868.947} C_VEL
LIN {X 0,Y 189.926,Z 287.089,A -85,B 0,C 180,E1 -22871.091,E2 -22871.091} C_VEL
LIN {X 0,Y 191.932,Z 289.021,A -85,B 0,C 180,E1 -22872.794,E2 -22872.794} C_VEL
LIN {X 0,Y 194.515,Z 292.677,A -85,B 0,C 180,E1 -22874.887,E2 -22874.887} C_VEL
LIN {X 0,Y 195.596,Z 293.921,A -85,B 0,C 180,E1 -22875.675,E2 -22875.675} C_VEL
LIN {X 0,Y 199.559,Z 299.436,A -85,B 0,C 180,E1 -22878.344,E2 -22878.344} C_VEL
LIN {X 0,Y 203.287,Z 305.365,A -85,B 0,C 180,E1 -22880.617,E2 -22880.617} C_VEL
LIN {X 0,Y 207.431,Z 312.43,A -85,B 0,C 180,E1 -22882.922,E2 -22882.922} C_VEL
LIN {X 0,Y 212.577,Z 322.123,A -85,B 0,C 180,E1 -22885.542,E2 -22885.542} C_VEL
LIN {X 0,Y 217.683,Z 333.205,A -85,B 0,C 180,E1 -22887.929,E2 -22887.929} C_VEL
LIN {X 0,Y 214.956,Z 370.371,A -85,B 0,C 180,E1 -22889.097,E2 -22889.097} C_VEL
LIN {X 0,Y 212.934,Z 383.689,A -85,B 0,C 180,E1 -22889.783,E2 -22889.783} C_VEL
LIN {X 0,Y 210.483,Z 395.361,A -85,B 0,C 180,E1 -22890.706,E2 -22890.706} C_VEL
LIN {X 0,Y 207.11,Z 407.257,A -85,B 0,C 180,E1 -22891.967,E2 -22891.967} C_VEL
LIN {X 0,Y 203.127,Z 418.652,A -85,B 0,C 180,E1 -22893.601,E2 -22893.601} C_VEL
LIN {X 0,Y 198.728,Z 429.207,A -85,B 0,C 180,E1 -22895.57,E2 -22895.57} C_VEL
LIN {X 0,Y 193.867,Z 439.225,A -85,B 0,C 180,E1 -22898.031,E2 -22898.031} C_VEL
LIN {X 0,Y 188.628,Z 448.514,A -85,B 0,C 180,E1 -22901.019,E2 -22901.019} C_VEL
LIN {X 0,Y 183.928,Z 455.968,A -85,B 0,C 180,E1 -22904.237,E2 -22904.237} C_VEL
LIN {X 0,Y 180.448,Z 460.968,A -85,B 0,C 180,E1 -22907.033,E2 -22907.033} C_VEL
LIN {X 0,Y 176.856,Z 465.679,A -85,B 0,C 180,E1 -22910.519,E2 -22910.519} C_VEL
LIN {X 0,Y 174.257,Z 468.871,A -85,B 0,C 180,E1 -22913.746,E2 -22913.746} C_VEL
LIN {X 0,Y 171.686,Z 471.552,A -85,B 0,C 180,E1 -22917.848,E2 -22917.848} C_VEL
LIN {X 0,Y 170.545,Z 472.552,A -85,B 0,C 180,E1 -22920.362,E2 -22920.362} C_VEL
LIN {X 0,Y 169.646,Z 473.117,A -85,B 0,C 180,E1 -22922.889,E2 -22922.889} C_VEL
LIN {X 0,Y 168.912,Z 473.135,A -85,B 0,C 180,E1 -22926.225,E2 -22926.225} C_VEL
LIN {X 0,Y 168.418,Z 472.083,A -85,B 0,C 180,E1 -22930.497,E2 -22930.497} C_VEL
LIN {X 0,Y 168.419,Z 470.457,A -85,B 0,C 180,E1 -22933.646,E2 -22933.646} C_VEL
LIN {X 0,Y 168.88,Z 467.053,A -85,B 0,C 180,E1 -22937.99,E2 -22937.99} C_VEL
LIN {X 0,Y 169.573,Z 462.952,A -85,B 0,C 180,E1 -22941.659,E2 -22941.659} C_VEL
LIN {X 0,Y 170.879,Z 456.62,A -85,B 0,C 180,E1 -22945.872,E2 -22945.872} C_VEL
LIN {X 0,Y 172.469,Z 449.721,A -85,B 0,C 180,E1 -22949.416,E2 -22949.416} C_VEL
LIN {X 0,Y 174.589,Z 441.117,A -85,B 0,C 180,E1 -22952.883,E2 -22952.883} C_VEL
LIN {X 0,Y 176.775,Z 432.178,A -85,B 0,C 180,E1 -22955.72,E2 -22955.72} C_VEL
LIN {X 0,Y 179.081,Z 422.469,A -85,B 0,C 180,E1 -22958.178,E2 -22958.178} C_VEL
LIN {X 0,Y 181.418,Z 411.766,A -85,B 0,C 180,E1 -22960.321,E2 -22960.321} C_VEL
LIN {X 0,Y 183.579,Z 399.874,A -85,B 0,C 180,E1 -22962.154,E2 -22962.154} C_VEL
LIN {X 0,Y 185.336,Z 387.523,A -85,B 0,C 180,E1 -22963.569,E2 -22963.569} C_VEL
LIN {X 0,Y 186.71,Z 374.872,A -85,B 0,C 180,E1 -22964.579,E2 -22964.579} C_VEL
LIN {X 0,Y 187.649,Z 360.647,A -85,B 0,C 180,E1 -22965.248,E2 -22965.248} C_VEL
LIN {X 0,Y 190.044,Z 308.311,A -85,B 0,C 180,E1 -22967.13,E2 -22967.13} C_VEL
LIN {X 0,Y 184.821,Z 293.145,A -85,B 0,C 180,E1 -22968.695,E2 -22968.695} C_VEL
LIN {X 0,Y 179.814,Z 281.195,A -85,B 0,C 180,E1 -22970.184,E2 -22970.184} C_VEL
LIN {X 0,Y 173.026,Z 269.197,A -85,B 0,C 180,E1 -22972.171,E2 -22972.171} C_VEL
LIN {X 0,Y 171.628,Z 266.469,A -85,B 0,C 180,E1 -22972.684,E2 -22972.684} C_VEL
LIN {X 0,Y 171.475,Z 265.682,A -85,B 0,C 180,E1 -22973.234,E2 -22973.234} C_VEL
LIN {X 0,Y 171.388,Z 265.578,A -85,B 0,C 180,E1 -22976.811,E2 -22976.811} C_VEL
LIN {X 0,Y 171.432,Z 265.616,A -85,B 0,C 180,E1 -22980.606,E2 -22980.606} C_VEL
LIN {X 0,Y 171.415,Z 265.613,A -85,B 0,C 180,E1 -22985.028,E2 -22985.028} C_VEL
LIN {X 0,Y 171.427,Z 265.632,A -85,B 0,C 180,E1 -22988.856,E2 -22988.856} C_VEL
LIN {X 0,Y 171.426,Z 265.611,A -85,B 0,C 180,E1 -22994.182,E2 -22994.182} C_VEL
LIN {X 0,Y 171.408,Z 265.611,A -85,B 0,C 180,E1 -22999.019,E2 -22999.019} C_VEL
LIN {X 0,Y 171.418,Z 265.592,A -85,B 0,C 180,E1 -23002.064,E2 -23002.064} C_VEL
LIN {X 0,Y 171.399,Z 265.63,A -85,B 0,C 180,E1 -23007.802,E2 -23007.802} C_VEL
LIN {X 0,Y 171.429,Z 265.589,A -85,B 0,C 180,E1 -23010.544,E2 -23010.544} C_VEL
LIN {X 0,Y 171.451,Z 265.61,A -85,B 0,C 180,E1 -23015.813,E2 -23015.813} C_VEL
LIN {X 0,Y 171.598,Z 265.594,A -85,B 0,C 180,E1 -23020.886,E2 -23020.886} C_VEL
LIN {X 0,Y 171.576,Z 265.555,A -85,B 0,C 180,E1 -23025.784,E2 -23025.784} C_VEL
LIN {X 0,Y 171.897,Z 265.57,A -85,B 0,C 180,E1 -23030.599,E2 -23030.599} C_VEL
LIN {X 0,Y 171.818,Z 265.542,A -85,B 0,C 180,E1 -23035.318,E2 -23035.318} C_VEL
LIN {X 0,Y 172.328,Z 265.475,A -85,B 0,C 180,E1 -23040.011,E2 -23040.011} C_VEL
LIN {X 0,Y 171.808,Z 265.583,A -85,B 0,C 180,E1 -23044.703,E2 -23044.703} C_VEL
LIN {X 0,Y 171.846,Z 265.529,A -85,B 0,C 180,E1 -23049.425,E2 -23049.425} C_VEL
LIN {X 0,Y 171.58,Z 265.603,A -85,B 0,C 180,E1 -23054.237,E2 -23054.237} C_VEL
LIN {X 0,Y 171.547,Z 265.582,A -85,B 0,C 180,E1 -23059.567,E2 -23059.567} C_VEL
LIN {X 0,Y 171.467,Z 265.629,A -85,B 0,C 180,E1 -23065.617,E2 -23065.617} C_VEL
LIN {X 0,Y 171.432,Z 265.604,A -85,B 0,C 180,E1 -23070.583,E2 -23070.583} C_VEL
LIN {X 0,Y 171.405,Z 265.63,A -85,B 0,C 180,E1 -23075.043,E2 -23075.043} C_VEL
LIN {X 0,Y 171.362,Z 265.628,A -85,B 0,C 180,E1 -23078.811,E2 -23078.811} C_VEL
LIN {X 0,Y 171.334,Z 265.586,A -85,B 0,C 180,E1 -23084.225,E2 -23084.225} C_VEL
LIN {X 0,Y 171.41,Z 265.796,A -85,B 0,C 180,E1 -23088.705,E2 -23088.705} C_VEL
LIN {X 0,Y 171.586,Z 266.666,A -85,B 0,C 180,E1 -23089.149,E2 -23089.149} C_VEL
LIN {X 0,Y 175.829,Z 274.908,A -85,B 0,C 180,E1 -23090.54,E2 -23090.54} C_VEL
LIN {X 0,Y 181.191,Z 287.136,A -85,B 0,C 180,E1 -23092.191,E2 -23092.191} C_VEL
LIN {X 0,Y 186.476,Z 301.269,A -85,B 0,C 180,E1 -23093.794,E2 -23093.794} C_VEL
LIN {X 0,Y 188.348,Z 307.261,A -85,B 0,C 180,E1 -23094.378,E2 -23094.378} C_VEL
LIN {X 0,Y 189.701,Z 320.091,A -85,B 0,C 180,E1 -23095.156,E2 -23095.156} C_VEL
LIN {X 0,Y 187.121,Z 374.883,A -85,B 0,C 180,E1 -23097.196,E2 -23097.196} C_VEL
LIN {X 0,Y 186.031,Z 385.527,A -85,B 0,C 180,E1 -23097.868,E2 -23097.868} C_VEL
LIN {X 0,Y 185.279,Z 389.29,A -85,B 0,C 180,E1 -23098.132,E2 -23098.132} C_VEL
LIN {X 0,Y 183.375,Z 394.78,A -85,B 0,C 180,E1 -23098.489,E2 -23098.489} C_VEL
LIN {X 0,Y 177.477,Z 407.034,A -85,B 0,C 180,E1 -23099.461,E2 -23099.461} C_VEL
LIN {X 0,Y 175.475,Z 412.256,A -85,B 0,C 180,E1 -23100.132,E2 -23100.132} C_VEL
LIN {X 0,Y 175.004,Z 413.953,A -85,B 0,C 180,E1 -23100.404,E2 -23100.404} C_VEL
LIN {X 0,Y 172.69,Z 424.364,A -85,B 0,C 180,E1 -23102.425,E2 -23102.425} C_VEL
LIN {X 0,Y 170.311,Z 434.622,A -85,B 0,C 180,E1 -23104.979,E2 -23104.979} C_VEL
LIN {X 0,Y 168.575,Z 441.432,A -85,B 0,C 180,E1 -23107.054,E2 -23107.054} C_VEL
LIN {X 0,Y 166.35,Z 450.05,A -85,B 0,C 180,E1 -23110.247,E2 -23110.247} C_VEL
LIN {X 0,Y 164.362,Z 457.72,A -85,B 0,C 180,E1 -23113.864,E2 -23113.864} C_VEL
LIN {X 0,Y 163.046,Z 463.879,A -85,B 0,C 180,E1 -23117.555,E2 -23117.555} C_VEL
LIN {X 0,Y 162.198,Z 468.734,A -85,B 0,C 180,E1 -23121.278,E2 -23121.278} C_VEL
LIN {X 0,Y 161.817,Z 472.44,A -85,B 0,C 180,E1 -23125.018,E2 -23125.018} C_VEL
LIN {X 0,Y 161.748,Z 474.778,A -85,B 0,C 180,E1 -23128.195,E2 -23128.195} C_VEL
LIN {X 0,Y 161.748,Z 476.586,A -85,B 0,C 180,E1 -23131.807,E2 -23131.807} C_VEL
LIN {X 0,Y 161.824,Z 477.428,A -85,B 0,C 180,E1 -23134.984,E2 -23134.984} C_VEL
LIN {X 0,Y 162.158,Z 477.674,A -85,B 0,C 180,E1 -23137.472,E2 -23137.472} C_VEL
LIN {X 0,Y 162.632,Z 477.528,A -85,B 0,C 180,E1 -23139.955,E2 -23139.955} C_VEL
LIN {X 0,Y 164.381,Z 476.028,A -85,B 0,C 180,E1 -23144.865,E2 -23144.865} C_VEL
LIN {X 0,Y 167.225,Z 472.984,A -85,B 0,C 180,E1 -23149.647,E2 -23149.647} C_VEL
LIN {X 0,Y 170.238,Z 469.552,A -85,B 0,C 180,E1 -23153.092,E2 -23153.092} C_VEL
LIN {X 0,Y 173.756,Z 465.072,A -85,B 0,C 180,E1 -23156.419,E2 -23156.419} C_VEL
LIN {X 0,Y 178.205,Z 458.71,A -85,B 0,C 180,E1 -23159.961,E2 -23159.961} C_VEL
LIN {X 0,Y 183.218,Z 451.018,A -85,B 0,C 180,E1 -23163.136,E2 -23163.136} C_VEL
LIN {X 0,Y 188.483,Z 441.975,A -85,B 0,C 180,E1 -23165.964,E2 -23165.964} C_VEL
LIN {X 0,Y 193.801,Z 431.536,A -85,B 0,C 180,E1 -23168.391,E2 -23168.391} C_VEL
LIN {X 0,Y 198.311,Z 420.967,A -85,B 0,C 180,E1 -23170.299,E2 -23170.299} C_VEL
LIN {X 0,Y 202.043,Z 410.753,A -85,B 0,C 180,E1 -23171.703,E2 -23171.703} C_VEL
LIN {X 0,Y 205.641,Z 398.589,A -85,B 0,C 180,E1 -23172.953,E2 -23172.953} C_VEL
LIN {X 0,Y 208.633,Z 384.934,A -85,B 0,C 180,E1 -23173.951,E2 -23173.951} C_VEL
LIN {X 0,Y 210.398,Z 372.691,A -85,B 0,C 180,E1 -23174.546,E2 -23174.546} C_VEL
LIN {X 0,Y 212.896,Z 339.403,A -85,B 0,C 180,E1 -23175.587,E2 -23175.587} C_VEL
LIN {X 0,Y 208.626,Z 329.187,A -85,B 0,C 180,E1 -23177.784,E2 -23177.784} C_VEL
LIN {X 0,Y 203.456,Z 318.712,A -85,B 0,C 180,E1 -23180.63,E2 -23180.63} C_VEL
LIN {X 0,Y 198.954,Z 310.647,A -85,B 0,C 180,E1 -23183.364,E2 -23183.364} C_VEL
LIN {X 0,Y 195.304,Z 304.688,A -85,B 0,C 180,E1 -23185.821,E2 -23185.821} C_VEL
LIN {X 0,Y 193.149,Z 301.136,A -85,B 0,C 180,E1 -23187.468,E2 -23187.468} C_VEL
LIN {X 0,Y 189.848,Z 296.165,A -85,B 0,C 180,E1 -23190.255,E2 -23190.255} C_VEL
LIN {X 0,Y 185.592,Z 290.16,A -85,B 0,C 180,E1 -23194.592,E2 -23194.592} C_VEL
LIN {X 0,Y 182.795,Z 287.266,A -85,B 0,C 180,E1 -23198.123,E2 -23198.123} C_VEL
LIN {X 0,Y 181.486,Z 284.684,A -85,B 0,C 180,E1 -23200.516,E2 -23200.516} C_VEL
LIN {X 0,Y 178.538,Z 282.232,A -85,B 0,C 180,E1 -23210.931,E2 -23210.931} C_VEL
LIN {X 0,Y 180.142,Z 283.463,A -85,B 0,C 180,E1 -23218.872,E2 -23218.872} C_VEL
LIN {X 0,Y 181.943,Z 284.768,A -85,B 0,C 180,E1 -23222.453,E2 -23222.453} C_VEL
LIN {X 0,Y 183.515,Z 287.822,A -85,B 0,C 180,E1 -23225.091,E2 -23225.091} C_VEL
LIN {X 0,Y 186.129,Z 290.182,A -85,B 0,C 180,E1 -23228.164,E2 -23228.164} C_VEL
LIN {X 0,Y 188.43,Z 293.856,A -85,B 0,C 180,E1 -23230.619,E2 -23230.619} C_VEL
LIN {X 0,Y 190.087,Z 295.543,A -85,B 0,C 180,E1 -23232.095,E2 -23232.095} C_VEL
LIN {X 0,Y 192.85,Z 299.387,A -85,B 0,C 180,E1 -23234.41,E2 -23234.41} C_VEL
LIN {X 0,Y 197.19,Z 305.501,A -85,B 0,C 180,E1 -23237.543,E2 -23237.543} C_VEL
LIN {X 0,Y 202.057,Z 313.54,A -85,B 0,C 180,E1 -23240.605,E2 -23240.605} C_VEL
LIN {X 0,Y 207.548,Z 323.789,A -85,B 0,C 180,E1 -23243.685,E2 -23243.685} C_VEL
LIN {X 0,Y 212.273,Z 334.006,A -85,B 0,C 180,E1 -23246.116,E2 -23246.116} C_VEL
LIN {X 0,Y 213.132,Z 336.075,A -85,B 0,C 180,E1 -23246.543,E2 -23246.543} C_VEL
LIN {X 0,Y 210.427,Z 370.619,A -85,B 0,C 180,E1 -23247.629,E2 -23247.629} C_VEL
LIN {X 0,Y 208.319,Z 383.95,A -85,B 0,C 180,E1 -23248.317,E2 -23248.317} C_VEL
LIN {X 0,Y 205.566,Z 396.484,A -85,B 0,C 180,E1 -23249.33,E2 -23249.33} C_VEL
LIN {X 0,Y 202.066,Z 408.086,A -85,B 0,C 180,E1 -23250.59,E2 -23250.59} C_VEL
LIN {X 0,Y 197.71,Z 419.958,A -85,B 0,C 180,E1 -23252.341,E2 -23252.341} C_VEL
LIN {X 0,Y 193.362,Z 429.789,A -85,B 0,C 180,E1 -23254.22,E2 -23254.22} C_VEL
LIN {X 0,Y 188.498,Z 439.335,A -85,B 0,C 180,E1 -23256.609,E2 -23256.609} C_VEL
LIN {X 0,Y 183.721,Z 447.48,A -85,B 0,C 180,E1 -23259.227,E2 -23259.227} C_VEL
LIN {X 0,Y 178.68,Z 455.201,A -85,B 0,C 180,E1 -23262.481,E2 -23262.481} C_VEL
LIN {X 0,Y 174.934,Z 460.339,A -85,B 0,C 180,E1 -23265.326,E2 -23265.326} C_VEL
LIN {X 0,Y 170.993,Z 465.247,A -85,B 0,C 180,E1 -23268.881,E2 -23268.881} C_VEL
LIN {X 0,Y 167.692,Z 469.016,A -85,B 0,C 180,E1 -23272.756,E2 -23272.756} C_VEL
LIN {X 0,Y 165.238,Z 471.42,A -85,B 0,C 180,E1 -23276.432,E2 -23276.432} C_VEL
LIN {X 0,Y 163.947,Z 472.488,A -85,B 0,C 180,E1 -23279.041,E2 -23279.041} C_VEL
LIN {X 0,Y 162.893,Z 473.128,A -85,B 0,C 180,E1 -23281.666,E2 -23281.666} C_VEL
LIN {X 0,Y 161.917,Z 473.234,A -85,B 0,C 180,E1 -23285.681,E2 -23285.681} C_VEL
LIN {X 0,Y 161.358,Z 472.353,A -85,B 0,C 180,E1 -23289.607,E2 -23289.607} C_VEL
LIN {X 0,Y 161.31,Z 470.572,A -85,B 0,C 180,E1 -23293.388,E2 -23293.388} C_VEL
LIN {X 0,Y 161.694,Z 467.586,A -85,B 0,C 180,E1 -23297.447,E2 -23297.447} C_VEL
LIN {X 0,Y 162.384,Z 463.625,A -85,B 0,C 180,E1 -23301.286,E2 -23301.286} C_VEL
LIN {X 0,Y 163.654,Z 457.523,A -85,B 0,C 180,E1 -23305.689,E2 -23305.689} C_VEL
LIN {X 0,Y 165.271,Z 450.795,A -85,B 0,C 180,E1 -23309.39,E2 -23309.39} C_VEL
LIN {X 0,Y 167.384,Z 442.439,A -85,B 0,C 180,E1 -23313.008,E2 -23313.008} C_VEL
LIN {X 0,Y 169.493,Z 434.39,A -85,B 0,C 180,E1 -23315.777,E2 -23315.777} C_VEL
LIN {X 0,Y 171.989,Z 424.415,A -85,B 0,C 180,E1 -23318.518,E2 -23318.518} C_VEL
LIN {X 0,Y 174.669,Z 412.663,A -85,B 0,C 180,E1 -23321.017,E2 -23321.017} C_VEL
LIN {X 0,Y 176.894,Z 401.075,A -85,B 0,C 180,E1 -23322.913,E2 -23322.913} C_VEL
LIN {X 0,Y 178.73,Z 389.066,A -85,B 0,C 180,E1 -23324.371,E2 -23324.371} C_VEL
LIN {X 0,Y 180.235,Z 376.084,A -85,B 0,C 180,E1 -23325.477,E2 -23325.477} C_VEL
LIN {X 0,Y 181.195,Z 363.515,A -85,B 0,C 180,E1 -23326.138,E2 -23326.138} C_VEL
LIN {X 0,Y 183.778,Z 309.653,A -85,B 0,C 180,E1 -23328.137,E2 -23328.137} C_VEL
LIN {X 0,Y 178.033,Z 293.321,A -85,B 0,C 180,E1 -23329.959,E2 -23329.959} C_VEL
LIN {X 0,Y 173.945,Z 283.907,A -85,B 0,C 180,E1 -23331.242,E2 -23331.242} C_VEL
LIN {X 0,Y 165.964,Z 270.124,A -85,B 0,C 180,E1 -23333.718,E2 -23333.718} C_VEL
LIN {X 0,Y 164.523,Z 267.194,A -85,B 0,C 180,E1 -23334.357,E2 -23334.357} C_VEL
LIN {X 0,Y 164.389,Z 266.524,A -85,B 0,C 180,E1 -23334.971,E2 -23334.971} C_VEL
LIN {X 0,Y 164.367,Z 266.508,A -85,B 0,C 180,E1 -23341.248,E2 -23341.248} C_VEL
LIN {X 0,Y 164.344,Z 266.5,A -85,B 0,C 180,E1 -23346.775,E2 -23346.775} C_VEL
LIN {X 0,Y 164.352,Z 266.501,A -85,B 0,C 180,E1 -23349.897,E2 -23349.897} C_VEL
LIN {X 0,Y 164.364,Z 266.483,A -85,B 0,C 180,E1 -23353.392,E2 -23353.392} C_VEL
LIN {X 0,Y 164.37,Z 266.511,A -85,B 0,C 180,E1 -23356.851,E2 -23356.851} C_VEL
LIN {X 0,Y 164.352,Z 266.474,A -85,B 0,C 180,E1 -23360.327,E2 -23360.327} C_VEL
LIN {X 0,Y 164.325,Z 266.5,A -85,B 0,C 180,E1 -23364.35,E2 -23364.35} C_VEL
LIN {X 0,Y 164.371,Z 266.487,A -85,B 0,C 180,E1 -23369.145,E2 -23369.145} C_VEL
LIN {X 0,Y 164.401,Z 266.47,A -85,B 0,C 180,E1 -23374.705,E2 -23374.705} C_VEL
LIN {X 0,Y 164.507,Z 266.485,A -85,B 0,C 180,E1 -23380.028,E2 -23380.028} C_VEL
LIN {X 0,Y 164.524,Z 266.43,A -85,B 0,C 180,E1 -23385.161,E2 -23385.161} C_VEL
LIN {X 0,Y 164.827,Z 266.45,A -85,B 0,C 180,E1 -23390.192,E2 -23390.192} C_VEL
LIN {X 0,Y 164.855,Z 266.444,A -85,B 0,C 180,E1 -23392.663,E2 -23392.663} C_VEL
LIN {X 0,Y 165.046,Z 266.365,A -85,B 0,C 180,E1 -23397.571,E2 -23397.571} C_VEL
LIN {X 0,Y 165.291,Z 266.35,A -85,B 0,C 180,E1 -23400.011,E2 -23400.011} C_VEL
LIN {X 0,Y 164.757,Z 266.461,A -85,B 0,C 180,E1 -23404.905,E2 -23404.905} C_VEL
LIN {X 0,Y 164.825,Z 266.426,A -85,B 0,C 180,E1 -23407.36,E2 -23407.36} C_VEL
LIN {X 0,Y 164.705,Z 266.418,A -85,B 0,C 180,E1 -23411.07,E2 -23411.07} C_VEL
LIN {X 0,Y 164.489,Z 266.487,A -85,B 0,C 180,E1 -23417.413,E2 -23417.413} C_VEL
LIN {X 0,Y 164.48,Z 266.459,A -85,B 0,C 180,E1 -23419.999,E2 -23419.999} C_VEL
LIN {X 0,Y 164.393,Z 266.511,A -85,B 0,C 180,E1 -23426.135,E2 -23426.135} C_VEL
LIN {X 0,Y 164.372,Z 266.488,A -85,B 0,C 180,E1 -23431.227,E2 -23431.227} C_VEL
LIN {X 0,Y 164.295,Z 266.5,A -85,B 0,C 180,E1 -23436.801,E2 -23436.801} C_VEL
LIN {X 0,Y 164.303,Z 266.52,A -85,B 0,C 180,E1 -23439.925,E2 -23439.925} C_VEL
LIN {X 0,Y 164.296,Z 266.469,A -85,B 0,C 180,E1 -23443.349,E2 -23443.349} C_VEL
LIN {X 0,Y 164.342,Z 266.743,A -85,B 0,C 180,E1 -23447.174,E2 -23447.174} C_VEL
LIN {X 0,Y 164.661,Z 267.963,A -85,B 0,C 180,E1 -23447.652,E2 -23447.652} C_VEL
LIN {X 0,Y 169.018,Z 275.645,A -85,B 0,C 180,E1 -23449.109,E2 -23449.109} C_VEL
LIN {X 0,Y 174.753,Z 288.23,A -85,B 0,C 180,E1 -23450.971,E2 -23450.971} C_VEL
LIN {X 0,Y 180.736,Z 304.275,A -85,B 0,C 180,E1 -23452.9,E2 -23452.9} C_VEL
LIN {X 0,Y 182.249,Z 309.259,A -85,B 0,C 180,E1 -23453.405,E2 -23453.405} C_VEL
LIN {X 0,Y 183.419,Z 322.403,A -85,B 0,C 180,E1 -23454.208,E2 -23454.208} C_VEL
LIN {X 0,Y 180.788,Z 374.599,A -85,B 0,C 180,E1 -23456.203,E2 -23456.203} C_VEL
LIN {X 0,Y 179.428,Z 387.482,A -85,B 0,C 180,E1 -23457.081,E2 -23457.081} C_VEL
LIN {X 0,Y 177.668,Z 400.153,A -85,B 0,C 180,E1 -23458.391,E2 -23458.391} C_VEL
LIN {X 0,Y 175.588,Z 411.39,A -85,B 0,C 180,E1 -23459.98,E2 -23459.98} C_VEL
LIN {X 0,Y 175.004,Z 413.953,A -85,B 0,C 180,E1 -23460.404,E2 -23460.404} C_VEL
LIN {X 0,Y 173.582,Z 417.372,A -85,B 0,C 180,E1 -23460.912,E2 -23460.912} C_VEL
LIN {X 0,Y 165.916,Z 427.58,A -85,B 0,C 180,E1 -23462.409,E2 -23462.409} C_VEL
LIN {X 0,Y 164.589,Z 430.667,A -85,B 0,C 180,E1 -23463.143,E2 -23463.143} C_VEL
LIN {X 0,Y 161.981,Z 439.962,A -85,B 0,C 180,E1 -23465.882,E2 -23465.882} C_VEL
LIN {X 0,Y 160.981,Z 444.603,A -85,B 0,C 180,E1 -23467.543,E2 -23467.543} C_VEL
LIN {X 0,Y 158.892,Z 452.039,A -85,B 0,C 180,E1 -23470.627,E2 -23470.627} C_VEL
LIN {X 0,Y 156.923,Z 459.335,A -85,B 0,C 180,E1 -23474.413,E2 -23474.413} C_VEL
LIN {X 0,Y 155.721,Z 465.15,A -85,B 0,C 180,E1 -23478.283,E2 -23478.283} C_VEL
LIN {X 0,Y 154.974,Z 469.698,A -85,B 0,C 180,E1 -23482.182,E2 -23482.182} C_VEL
LIN {X 0,Y 154.74,Z 472.083,A -85,B 0,C 180,E1 -23484.789,E2 -23484.789} C_VEL
LIN {X 0,Y 154.673,Z 474.902,A -85,B 0,C 180,E1 -23488.829,E2 -23488.829} C_VEL
LIN {X 0,Y 154.656,Z 476.608,A -85,B 0,C 180,E1 -23492.605,E2 -23492.605} C_VEL
LIN {X 0,Y 155.097,Z 477.555,A -85,B 0,C 180,E1 -23497.814,E2 -23497.814} C_VEL
LIN {X 0,Y 155.615,Z 477.462,A -85,B 0,C 180,E1 -23500.409,E2 -23500.409} C_VEL
LIN {X 0,Y 156.414,Z 476.965,A -85,B 0,C 180,E1 -23502.984,E2 -23502.984} C_VEL
LIN {X 0,Y 158.849,Z 474.782,A -85,B 0,C 180,E1 -23508.042,E2 -23508.042} C_VEL
LIN {X 0,Y 161.558,Z 472.086,A -85,B 0,C 180,E1 -23511.702,E2 -23511.702} C_VEL
LIN {X 0,Y 164.92,Z 468.402,A -85,B 0,C 180,E1 -23515.224,E2 -23515.224} C_VEL
LIN {X 0,Y 168.796,Z 463.638,A -85,B 0,C 180,E1 -23518.609,E2 -23518.609} C_VEL
LIN {X 0,Y 173.151,Z 457.657,A -85,B 0,C 180,E1 -23521.848,E2 -23521.848} C_VEL
LIN {X 0,Y 178.223,Z 450.226,A -85,B 0,C 180,E1 -23524.876,E2 -23524.876} C_VEL
LIN {X 0,Y 182.833,Z 442.664,A -85,B 0,C 180,E1 -23527.26,E2 -23527.26} C_VEL
LIN {X 0,Y 187.802,Z 433.525,A -85,B 0,C 180,E1 -23529.508,E2 -23529.508} C_VEL
LIN {X 0,Y 192.451,Z 423.416,A -85,B 0,C 180,E1 -23531.445,E2 -23531.445} C_VEL
LIN {X 0,Y 196.858,Z 412.229,A -85,B 0,C 180,E1 -23533.062,E2 -23533.062} C_VEL
LIN {X 0,Y 200.285,Z 401.635,A -85,B 0,C 180,E1 -23534.22,E2 -23534.22} C_VEL
LIN {X 0,Y 203.463,Z 388.956,A -85,B 0,C 180,E1 -23535.246,E2 -23535.246} C_VEL
LIN {X 0,Y 205.763,Z 375.189,A -85,B 0,C 180,E1 -23535.992,E2 -23535.992} C_VEL
LIN {X 0,Y 207.886,Z 350.183,A -85,B 0,C 180,E1 -23536.809,E2 -23536.809} C_VEL
LIN {X 0,Y 208.498,Z 342.095,A -85,B 0,C 180,E1 -23537.057,E2 -23537.057} C_VEL
LIN {X 0,Y 204.905,Z 333.386,A -85,B 0,C 180,E1 -23539.038,E2 -23539.038} C_VEL
LIN {X 0,Y 200.306,Z 323.793,A -85,B 0,C 180,E1 -23541.742,E2 -23541.742} C_VEL
LIN {X 0,Y 196.34,Z 316.399,A -85,B 0,C 180,E1 -23544.304,E2 -23544.304} C_VEL
LIN {X 0,Y 192.984,Z 310.683,A -85,B 0,C 180,E1 -23546.723,E2 -23546.723} C_VEL
LIN {X 0,Y 190.947,Z 307.168,A -85,B 0,C 180,E1 -23548.379,E2 -23548.379} C_VEL
LIN {X 0,Y 187.838,Z 302.324,A -85,B 0,C 180,E1 -23551.168,E2 -23551.168} C_VEL
LIN {X 0,Y 184.027,Z 296.744,A -85,B 0,C 180,E1 -23555.294,E2 -23555.294} C_VEL
LIN {X 0,Y 181.661,Z 294.251,A -85,B 0,C 180,E1 -23558.427,E2 -23558.427} C_VEL
LIN {X 0,Y 180.397,Z 291.654,A -85,B 0,C 180,E1 -23560.856,E2 -23560.856} C_VEL
LIN {X 0,Y 177.648,Z 289.285,A -85,B 0,C 180,E1 -23570.885,E2 -23570.885} C_VEL
LIN {X 0,Y 179.254,Z 290.499,A -85,B 0,C 180,E1 -23578.867,E2 -23578.867} C_VEL
LIN {X 0,Y 180.736,Z 291.657,A -85,B 0,C 180,E1 -23581.938,E2 -23581.938} C_VEL
LIN {X 0,Y 182.487,Z 294.974,A -85,B 0,C 180,E1 -23584.978,E2 -23584.978} C_VEL
LIN {X 0,Y 184.603,Z 296.94,A -85,B 0,C 180,E1 -23587.553,E2 -23587.553} C_VEL
LIN {X 0,Y 187.143,Z 300.842,A -85,B 0,C 180,E1 -23590.334,E2 -23590.334} C_VEL
LIN {X 0,Y 188.404,Z 302.247,A -85,B 0,C 180,E1 -23591.505,E2 -23591.505} C_VEL
LIN {X 0,Y 191.804,Z 307.146,A -85,B 0,C 180,E1 -23594.43,E2 -23594.43} C_VEL
LIN {X 0,Y 194.899,Z 311.71,A -85,B 0,C 180,E1 -23596.756,E2 -23596.756} C_VEL
LIN {X 0,Y 199.433,Z 319.485,A -85,B 0,C 180,E1 -23599.76,E2 -23599.76} C_VEL
LIN {X 0,Y 204.525,Z 329.399,A -85,B 0,C 180,E1 -23602.777,E2 -23602.777} C_VEL
LIN {X 0,Y 208.717,Z 338.797,A -85,B 0,C 180,E1 -23605.064,E2 -23605.064} C_VEL
LIN {X 0,Y 206.111,Z 370.739,A -85,B 0,C 180,E1 -23606.076,E2 -23606.076} C_VEL
LIN {X 0,Y 203.869,Z 384.443,A -85,B 0,C 180,E1 -23606.792,E2 -23606.792} C_VEL
LIN {X 0,Y 201.065,Z 396.591,A -85,B 0,C 180,E1 -23607.776,E2 -23607.776} C_VEL
LIN {X 0,Y 197.149,Z 409.007,A -85,B 0,C 180,E1 -23609.145,E2 -23609.145} C_VEL
LIN {X 0,Y 192.485,Z 421.029,A -85,B 0,C 180,E1 -23610.957,E2 -23610.957} C_VEL
LIN {X 0,Y 187.568,Z 431.401,A -85,B 0,C 180,E1 -23613.031,E2 -23613.031} C_VEL
LIN {X 0,Y 182.79,Z 440.254,A -85,B 0,C 180,E1 -23615.345,E2 -23615.345} C_VEL
LIN {X 0,Y 177.135,Z 449.314,A -85,B 0,C 180,E1 -23618.408,E2 -23618.408} C_VEL
LIN {X 0,Y 171.909,Z 456.678,A -85,B 0,C 180,E1 -23621.792,E2 -23621.792} C_VEL
LIN {X 0,Y 166.911,Z 462.934,A -85,B 0,C 180,E1 -23625.691,E2 -23625.691} C_VEL
LIN {X 0,Y 162.871,Z 467.446,A -85,B 0,C 180,E1 -23629.664,E2 -23629.664} C_VEL
LIN {X 0,Y 160.749,Z 469.575,A -85,B 0,C 180,E1 -23632.259,E2 -23632.259} C_VEL
LIN {X 0,Y 158.923,Z 471.242,A -85,B 0,C 180,E1 -23634.907,E2 -23634.907} C_VEL
LIN {X 0,Y 157.188,Z 472.584,A -85,B 0,C 180,E1 -23638.132,E2 -23638.132} C_VEL
LIN {X 0,Y 155.33,Z 473.417,A -85,B 0,C 180,E1 -23643.098,E2 -23643.098} C_VEL
LIN {X 0,Y 154.78,Z 473.252,A -85,B 0,C 180,E1 -23645.879,E2 -23645.879} C_VEL
LIN {X 0,Y 154.33,Z 472.623,A -85,B 0,C 180,E1 -23648.634,E2 -23648.634} C_VEL
LIN {X 0,Y 154.204,Z 470.687,A -85,B 0,C 180,E1 -23653.106,E2 -23653.106} C_VEL
LIN {X 0,Y 154.713,Z 466.989,A -85,B 0,C 180,E1 -23658.204,E2 -23658.204} C_VEL
LIN {X 0,Y 155.471,Z 462.794,A -85,B 0,C 180,E1 -23662.205,E2 -23662.205} C_VEL
LIN {X 0,Y 156.663,Z 457.392,A -85,B 0,C 180,E1 -23666.141,E2 -23666.141} C_VEL
LIN {X 0,Y 158.368,Z 450.614,A -85,B 0,C 180,E1 -23669.999,E2 -23669.999} C_VEL
LIN {X 0,Y 160.616,Z 442.198,A -85,B 0,C 180,E1 -23673.762,E2 -23673.762} C_VEL
LIN {X 0,Y 163.015,Z 433.284,A -85,B 0,C 180,E1 -23676.886,E2 -23676.886} C_VEL
LIN {X 0,Y 165.717,Z 422.797,A -85,B 0,C 180,E1 -23679.766,E2 -23679.766} C_VEL
LIN {X 0,Y 168.261,Z 412.117,A -85,B 0,C 180,E1 -23682.054,E2 -23682.054} C_VEL
LIN {X 0,Y 170.613,Z 400.282,A -85,B 0,C 180,E1 -23684.004,E2 -23684.004} C_VEL
LIN {X 0,Y 172.499,Z 388.009,A -85,B 0,C 180,E1 -23685.507,E2 -23685.507} C_VEL
LIN {X 0,Y 174.093,Z 374.7,A -85,B 0,C 180,E1 -23686.626,E2 -23686.626} C_VEL
LIN {X 0,Y 175.065,Z 360.527,A -85,B 0,C 180,E1 -23687.322,E2 -23687.322} C_VEL
LIN {X 0,Y 177.62,Z 311.487,A -85,B 0,C 180,E1 -23689.175,E2 -23689.175} C_VEL
LIN {X 0,Y 172.22,Z 295.946,A -85,B 0,C 180,E1 -23691.005,E2 -23691.005} C_VEL
LIN {X 0,Y 168.56,Z 287.555,A -85,B 0,C 180,E1 -23692.22,E2 -23692.22} C_VEL
LIN {X 0,Y 161.18,Z 274.689,A -85,B 0,C 180,E1 -23694.646,E2 -23694.646} C_VEL
LIN {X 0,Y 158.883,Z 270.933,A -85,B 0,C 180,E1 -23695.449,E2 -23695.449} C_VEL
LIN {X 0,Y 157.454,Z 268.052,A -85,B 0,C 180,E1 -23696.129,E2 -23696.129} C_VEL
LIN {X 0,Y 157.299,Z 267.413,A -85,B 0,C 180,E1 -23696.704,E2 -23696.704} C_VEL
LIN {X 0,Y 157.288,Z 267.395,A -85,B 0,C 180,E1 -23702.423,E2 -23702.423} C_VEL
LIN {X 0,Y 157.318,Z 267.372,A -85,B 0,C 180,E1 -23706.497,E2 -23706.497} C_VEL
LIN {X 0,Y 157.27,Z 267.363,A -85,B 0,C 180,E1 -23712.09,E2 -23712.09} C_VEL
LIN {X 0,Y 157.287,Z 267.389,A -85,B 0,C 180,E1 -23715.635,E2 -23715.635} C_VEL
LIN {X 0,Y 157.267,Z 267.352,A -85,B 0,C 180,E1 -23721.288,E2 -23721.288} C_VEL
LIN {X 0,Y 157.272,Z 267.379,A -85,B 0,C 180,E1 -23724.5,E2 -23724.5} C_VEL
LIN {X 0,Y 157.274,Z 267.386,A -85,B 0,C 180,E1 -23728.105,E2 -23728.105} C_VEL
LIN {X 0,Y 157.304,Z 267.34,A -85,B 0,C 180,E1 -23733.477,E2 -23733.477} C_VEL
LIN {X 0,Y 157.433,Z 267.37,A -85,B 0,C 180,E1 -23739.627,E2 -23739.627} C_VEL
LIN {X 0,Y 157.455,Z 267.309,A -85,B 0,C 180,E1 -23744.479,E2 -23744.479} C_VEL
LIN {X 0,Y 157.741,Z 267.328,A -85,B 0,C 180,E1 -23749.746,E2 -23749.746} C_VEL
LIN {X 0,Y 157.814,Z 267.324,A -85,B 0,C 180,E1 -23752.334,E2 -23752.334} C_VEL
LIN {X 0,Y 158.253,Z 267.225,A -85,B 0,C 180,E1 -23760.011,E2 -23760.011} C_VEL
LIN {X 0,Y 157.763,Z 267.298,A -85,B 0,C 180,E1 -23767.691,E2 -23767.691} C_VEL
LIN {X 0,Y 157.64,Z 267.298,A -85,B 0,C 180,E1 -23771.246,E2 -23771.246} C_VEL
LIN {X 0,Y 157.459,Z 267.371,A -85,B 0,C 180,E1 -23775.545,E2 -23775.545} C_VEL
LIN {X 0,Y 157.375,Z 267.341,A -85,B 0,C 180,E1 -23780.943,E2 -23780.943} C_VEL
LIN {X 0,Y 157.32,Z 267.387,A -85,B 0,C 180,E1 -23786.69,E2 -23786.69} C_VEL
LIN {X 0,Y 157.281,Z 267.385,A -85,B 0,C 180,E1 -23792.438,E2 -23792.438} C_VEL
LIN {X 0,Y 157.273,Z 267.376,A -85,B 0,C 180,E1 -23796.453,E2 -23796.453} C_VEL
LIN {X 0,Y 157.206,Z 267.368,A -85,B 0,C 180,E1 -23802.125,E2 -23802.125} C_VEL
LIN {X 0,Y 157.211,Z 267.563,A -85,B 0,C 180,E1 -23805.285,E2 -23805.285} C_VEL
LIN {X 0,Y 157.5,Z 268.676,A -85,B 0,C 180,E1 -23805.842,E2 -23805.842} C_VEL
LIN {X 0,Y 159.095,Z 271.329,A -85,B 0,C 180,E1 -23806.463,E2 -23806.463} C_VEL
LIN {X 0,Y 163.96,Z 279.832,A -85,B 0,C 180,E1 -23808.152,E2 -23808.152} C_VEL
LIN {X 0,Y 169.22,Z 291.48,A -85,B 0,C 180,E1 -23809.96,E2 -23809.96} C_VEL
LIN {X 0,Y 174.91,Z 306.963,A -85,B 0,C 180,E1 -23811.917,E2 -23811.917} C_VEL
LIN {X 0,Y 176.22,Z 311.453,A -85,B 0,C 180,E1 -23812.389,E2 -23812.389} C_VEL
LIN {X 0,Y 177.229,Z 322.227,A -85,B 0,C 180,E1 -23813.093,E2 -23813.093} C_VEL
LIN {X 0,Y 174.5,Z 374.402,A -85,B 0,C 180,E1 -23815.142,E2 -23815.142} C_VEL
LIN {X 0,Y 173.072,Z 387.489,A -85,B 0,C 180,E1 -23816.059,E2 -23816.059} C_VEL
LIN {X 0,Y 171.246,Z 400.132,A -85,B 0,C 180,E1 -23817.409,E2 -23817.409} C_VEL
LIN {X 0,Y 169.076,Z 411.346,A -85,B 0,C 180,E1 -23819.044,E2 -23819.044} C_VEL
LIN {X 0,Y 166.983,Z 420.373,A -85,B 0,C 180,E1 -23820.708,E2 -23820.708} C_VEL
LIN {X 0,Y 164.589,Z 430.667,A -85,B 0,C 180,E1 -23823.143,E2 -23823.143} C_VEL
LIN {X 0,Y 162.911,Z 435.223,A -85,B 0,C 180,E1 -23824.355,E2 -23824.355} C_VEL
LIN {X 0,Y 158.333,Z 442.148,A -85,B 0,C 180,E1 -23826.305,E2 -23826.305} C_VEL
LIN {X 0,Y 153.675,Z 448.494,A -85,B 0,C 180,E1 -23828.529,E2 -23828.529} C_VEL
LIN {X 0,Y 151.922,Z 452.129,A -85,B 0,C 180,E1 -23830.137,E2 -23830.137} C_VEL
LIN {X 0,Y 149.803,Z 459.79,A -85,B 0,C 180,E1 -23834.351,E2 -23834.351} C_VEL
LIN {X 0,Y 148.413,Z 466.291,A -85,B 0,C 180,E1 -23839.082,E2 -23839.082} C_VEL
LIN {X 0,Y 147.772,Z 470.549,A -85,B 0,C 180,E1 -23843.172,E2 -23843.172} C_VEL
LIN {X 0,Y 147.579,Z 473.714,A -85,B 0,C 180,E1 -23847.271,E2 -23847.271} C_VEL
LIN {X 0,Y 147.621,Z 475.575,A -85,B 0,C 180,E1 -23850.614,E2 -23850.614} C_VEL
LIN {X 0,Y 147.674,Z 477.114,A -85,B 0,C 180,E1 -23855.463,E2 -23855.463} C_VEL
LIN {X 0,Y 148.051,Z 477.437,A -85,B 0,C 180,E1 -23858.188,E2 -23858.188} C_VEL
LIN {X 0,Y 149.495,Z 476.951,A -85,B 0,C 180,E1 -23863.596,E2 -23863.596} C_VEL
LIN {X 0,Y 152.09,Z 474.859,A -85,B 0,C 180,E1 -23868.873,E2 -23868.873} C_VEL
LIN {X 0,Y 156.086,Z 471.179,A -85,B 0,C 180,E1 -23873.907,E2 -23873.907} C_VEL
LIN {X 0,Y 159.817,Z 467.229,A -85,B 0,C 180,E1 -23877.5,E2 -23877.5} C_VEL
LIN {X 0,Y 164.575,Z 461.508,A -85,B 0,C 180,E1 -23881.325,E2 -23881.325} C_VEL
LIN {X 0,Y 169.735,Z 454.659,A -85,B 0,C 180,E1 -23884.704,E2 -23884.704} C_VEL
LIN {X 0,Y 175.346,Z 446.541,A -85,B 0,C 180,E1 -23887.679,E2 -23887.679} C_VEL
LIN {X 0,Y 180.334,Z 438.269,A -85,B 0,C 180,E1 -23890.02,E2 -23890.02} C_VEL
LIN {X 0,Y 185.594,Z 428.129,A -85,B 0,C 180,E1 -23892.234,E2 -23892.234} C_VEL
LIN {X 0,Y 190.686,Z 416.697,A -85,B 0,C 180,E1 -23894.081,E2 -23894.081} C_VEL
LIN {X 0,Y 194.761,Z 405.476,A -85,B 0,C 180,E1 -23895.454,E2 -23895.454} C_VEL
LIN {X 0,Y 198.057,Z 393.875,A -85,B 0,C 180,E1 -23896.513,E2 -23896.513} C_VEL
LIN {X 0,Y 200.812,Z 380.515,A -85,B 0,C 180,E1 -23897.359,E2 -23897.359} C_VEL
LIN {X 0,Y 202.475,Z 366.979,A -85,B 0,C 180,E1 -23897.918,E2 -23897.918} C_VEL
LIN {X 0,Y 204.205,Z 344.713,A -85,B 0,C 180,E1 -23898.61,E2 -23898.61} C_VEL
LIN {X 0,Y 200.717,Z 336.216,A -85,B 0,C 180,E1 -23900.688,E2 -23900.688} C_VEL
LIN {X 0,Y 196.15,Z 326.588,A -85,B 0,C 180,E1 -23903.621,E2 -23903.621} C_VEL
LIN {X 0,Y 191.94,Z 318.675,A -85,B 0,C 180,E1 -23906.676,E2 -23906.676} C_VEL
LIN {X 0,Y 188.792,Z 313.236,A -85,B 0,C 180,E1 -23909.309,E2 -23909.309} C_VEL
LIN {X 0,Y 186.086,Z 308.799,A -85,B 0,C 180,E1 -23911.887,E2 -23911.887} C_VEL
LIN {X 0,Y 182.608,Z 303.493,A -85,B 0,C 180,E1 -23915.854,E2 -23915.854} C_VEL
LIN {X 0,Y 180.37,Z 300.981,A -85,B 0,C 180,E1 -23919.014,E2 -23919.014} C_VEL
LIN {X 0,Y 179.19,Z 298.561,A -85,B 0,C 180,E1 -23921.416,E2 -23921.416} C_VEL
LIN {X 0,Y 176.759,Z 296.34,A -85,B 0,C 180,E1 -23930.839,E2 -23930.839} C_VEL
LIN {X 0,Y 177.916,Z 297.316,A -85,B 0,C 180,E1 -23937.726,E2 -23937.726} C_VEL
LIN {X 0,Y 179.521,Z 298.509,A -85,B 0,C 180,E1 -23941.388,E2 -23941.388} C_VEL
LIN {X 0,Y 181.358,Z 301.976,A -85,B 0,C 180,E1 -23944.722,E2 -23944.722} C_VEL
LIN {X 0,Y 183.152,Z 303.747,A -85,B 0,C 180,E1 -23946.994,E2 -23946.994} C_VEL
LIN {X 0,Y 185.748,Z 307.683,A -85,B 0,C 180,E1 -23949.932,E2 -23949.932} C_VEL
LIN {X 0,Y 186.802,Z 309.093,A -85,B 0,C 180,E1 -23950.97,E2 -23950.97} C_VEL
LIN {X 0,Y 189.877,Z 313.608,A -85,B 0,C 180,E1 -23953.729,E2 -23953.729} C_VEL
LIN {X 0,Y 192.618,Z 317.818,A -85,B 0,C 180,E1 -23955.905,E2 -23955.905} C_VEL
LIN {X 0,Y 197.123,Z 325.928,A -85,B 0,C 180,E1 -23959.07,E2 -23959.07} C_VEL
LIN {X 0,Y 201.687,Z 335.277,A -85,B 0,C 180,E1 -23961.921,E2 -23961.921} C_VEL
LIN {X 0,Y 204.481,Z 341.778,A -85,B 0,C 180,E1 -23963.552,E2 -23963.552} C_VEL
LIN {X 0,Y 201.938,Z 371.085,A -85,B 0,C 180,E1 -23964.475,E2 -23964.475} C_VEL
LIN {X 0,Y 199.668,Z 384.456,A -85,B 0,C 180,E1 -23965.167,E2 -23965.167} C_VEL
LIN {X 0,Y 196.69,Z 396.844,A -85,B 0,C 180,E1 -23966.164,E2 -23966.164} C_VEL
LIN {X 0,Y 192.986,Z 408.312,A -85,B 0,C 180,E1 -23967.417,E2 -23967.417} C_VEL
LIN {X 0,Y 188.383,Z 419.922,A -85,B 0,C 180,E1 -23969.133,E2 -23969.133} C_VEL
LIN {X 0,Y 183.556,Z 429.948,A -85,B 0,C 180,E1 -23971.051,E2 -23971.051} C_VEL
LIN {X 0,Y 178.147,Z 439.616,A -85,B 0,C 180,E1 -23973.512,E2 -23973.512} C_VEL
LIN {X 0,Y 172.514,Z 448.335,A -85,B 0,C 180,E1 -23976.429,E2 -23976.429} C_VEL
LIN {X 0,Y 167.379,Z 455.33,A -85,B 0,C 180,E1 -23979.51,E2 -23979.51} C_VEL
LIN {X 0,Y 162.784,Z 460.941,A -85,B 0,C 180,E1 -23982.78,E2 -23982.78} C_VEL
LIN {X 0,Y 158.398,Z 465.735,A -85,B 0,C 180,E1 -23986.549,E2 -23986.549} C_VEL
LIN {X 0,Y 154.779,Z 469.303,A -85,B 0,C 180,E1 -23990.528,E2 -23990.528} C_VEL
LIN {X 0,Y 152.709,Z 471.04,A -85,B 0,C 180,E1 -23993.252,E2 -23993.252} C_VEL
LIN {X 0,Y 150.39,Z 472.711,A -85,B 0,C 180,E1 -23997.238,E2 -23997.238} C_VEL
LIN {X 0,Y 148.593,Z 473.488,A -85,B 0,C 180,E1 -24001.772,E2 -24001.772} C_VEL
LIN {X 0,Y 147.882,Z 473.418,A -85,B 0,C 180,E1 -24004.676,E2 -24004.676} C_VEL
LIN {X 0,Y 147.366,Z 472.892,A -85,B 0,C 180,E1 -24007.571,E2 -24007.571} C_VEL
LIN {X 0,Y 147.089,Z 470.793,A -85,B 0,C 180,E1 -24012.814,E2 -24012.814} C_VEL
LIN {X 0,Y 147.524,Z 467.539,A -85,B 0,C 180,E1 -24017.62,E2 -24017.62} C_VEL
LIN {X 0,Y 148.28,Z 463.495,A -85,B 0,C 180,E1 -24021.825,E2 -24021.825} C_VEL
LIN {X 0,Y 149.713,Z 457.258,A -85,B 0,C 180,E1 -24026.635,E2 -24026.635} C_VEL
LIN {X 0,Y 151.511,Z 450.43,A -85,B 0,C 180,E1 -24030.664,E2 -24030.664} C_VEL
LIN {X 0,Y 153.883,Z 441.95,A -85,B 0,C 180,E1 -24034.583,E2 -24034.583} C_VEL
LIN {X 0,Y 156.335,Z 433.188,A -85,B 0,C 180,E1 -24037.75,E2 -24037.75} C_VEL
LIN {X 0,Y 158.956,Z 423.551,A -85,B 0,C 180,E1 -24040.508,E2 -24040.508} C_VEL
LIN {X 0,Y 161.577,Z 413.017,A -85,B 0,C 180,E1 -24042.88,E2 -24042.88} C_VEL
LIN {X 0,Y 164.019,Z 401.466,A -85,B 0,C 180,E1 -24044.897,E2 -24044.897} C_VEL
LIN {X 0,Y 165.984,Z 389.554,A -85,B 0,C 180,E1 -24046.448,E2 -24046.448} C_VEL
LIN {X 0,Y 167.715,Z 375.908,A -85,B 0,C 180,E1 -24047.673,E2 -24047.673} C_VEL
LIN {X 0,Y 168.748,Z 362.84,A -85,B 0,C 180,E1 -24048.38,E2 -24048.38} C_VEL
LIN {X 0,Y 171.396,Z 312.765,A -85,B 0,C 180,E1 -24050.338,E2 -24050.338} C_VEL
LIN {X 0,Y 165.464,Z 296.092,A -85,B 0,C 180,E1 -24052.473,E2 -24052.473} C_VEL
LIN {X 0,Y 162.101,Z 289.161,A -85,B 0,C 180,E1 -24053.63,E2 -24053.63} C_VEL
LIN {X 0,Y 154.45,Z 275.888,A -85,B 0,C 180,E1 -24056.373,E2 -24056.373} C_VEL
LIN {X 0,Y 152.117,Z 272.266,A -85,B 0,C 180,E1 -24057.261,E2 -24057.261} C_VEL
LIN {X 0,Y 150.535,Z 269.668,A -85,B 0,C 180,E1 -24057.925,E2 -24057.925} C_VEL
LIN {X 0,Y 150.231,Z 268.502,A -85,B 0,C 180,E1 -24058.414,E2 -24058.414} C_VEL
LIN {X 0,Y 150.203,Z 268.26,A -85,B 0,C 180,E1 -24060.976,E2 -24060.976} C_VEL
LIN {X 0,Y 150.197,Z 268.258,A -85,B 0,C 180,E1 -24064.158,E2 -24064.158} C_VEL
LIN {X 0,Y 150.242,Z 268.263,A -85,B 0,C 180,E1 -24067.452,E2 -24067.452} C_VEL
LIN {X 0,Y 150.211,Z 268.244,A -85,B 0,C 180,E1 -24071.552,E2 -24071.552} C_VEL
LIN {X 0,Y 150.262,Z 268.261,A -85,B 0,C 180,E1 -24075.466,E2 -24075.466} C_VEL
LIN {X 0,Y 150.212,Z 268.246,A -85,B 0,C 180,E1 -24079.097,E2 -24079.097} C_VEL
LIN {X 0,Y 150.216,Z 268.234,A -85,B 0,C 180,E1 -24082.688,E2 -24082.688} C_VEL
LIN {X 0,Y 150.198,Z 268.274,A -85,B 0,C 180,E1 -24087.376,E2 -24087.376} C_VEL
LIN {X 0,Y 150.226,Z 268.217,A -85,B 0,C 180,E1 -24092.73,E2 -24092.73} C_VEL
LIN {X 0,Y 150.376,Z 268.251,A -85,B 0,C 180,E1 -24099.18,E2 -24099.18} C_VEL
LIN {X 0,Y 150.366,Z 268.194,A -85,B 0,C 180,E1 -24103.727,E2 -24103.727} C_VEL
LIN {X 0,Y 150.655,Z 268.205,A -85,B 0,C 180,E1 -24109.258,E2 -24109.258} C_VEL
LIN {X 0,Y 150.75,Z 268.205,A -85,B 0,C 180,E1 -24111.973,E2 -24111.973} C_VEL
LIN {X 0,Y 151.214,Z 268.1,A -85,B 0,C 180,E1 -24120.012,E2 -24120.012} C_VEL
LIN {X 0,Y 150.685,Z 268.173,A -85,B 0,C 180,E1 -24128.055,E2 -24128.055} C_VEL
LIN {X 0,Y 150.58,Z 268.178,A -85,B 0,C 180,E1 -24131.447,E2 -24131.447} C_VEL
LIN {X 0,Y 150.368,Z 268.254,A -85,B 0,C 180,E1 -24136.298,E2 -24136.298} C_VEL
LIN {X 0,Y 150.357,Z 268.214,A -85,B 0,C 180,E1 -24140.801,E2 -24140.801} C_VEL
LIN {X 0,Y 150.25,Z 268.259,A -85,B 0,C 180,E1 -24147.288,E2 -24147.288} C_VEL
LIN {X 0,Y 150.222,Z 268.266,A -85,B 0,C 180,E1 -24152.638,E2 -24152.638} C_VEL
LIN {X 0,Y 150.183,Z 268.257,A -85,B 0,C 180,E1 -24157.483,E2 -24157.483} C_VEL
LIN {X 0,Y 150.144,Z 268.359,A -85,B 0,C 180,E1 -24163.136,E2 -24163.136} C_VEL
LIN {X 0,Y 150.369,Z 269.284,A -85,B 0,C 180,E1 -24163.787,E2 -24163.787} C_VEL
LIN {X 0,Y 151.964,Z 272.158,A -85,B 0,C 180,E1 -24164.52,E2 -24164.52} C_VEL
LIN {X 0,Y 157.404,Z 281.006,A -85,B 0,C 180,E1 -24166.562,E2 -24166.562} C_VEL
LIN {X 0,Y 161.734,Z 289.959,A -85,B 0,C 180,E1 -24168.158,E2 -24168.158} C_VEL
LIN {X 0,Y 167.195,Z 303.999,A -85,B 0,C 180,E1 -24170.155,E2 -24170.155} C_VEL
LIN {X 0,Y 170.25,Z 313.437,A -85,B 0,C 180,E1 -24171.291,E2 -24171.291} C_VEL
LIN {X 0,Y 171.061,Z 323.45,A -85,B 0,C 180,E1 -24171.957,E2 -24171.957} C_VEL
LIN {X 0,Y 168.257,Z 374.463,A -85,B 0,C 180,E1 -24174.018,E2 -24174.018} C_VEL
LIN {X 0,Y 166.769,Z 387.492,A -85,B 0,C 180,E1 -24174.959,E2 -24174.959} C_VEL
LIN {X 0,Y 164.866,Z 400.105,A -85,B 0,C 180,E1 -24176.347,E2 -24176.347} C_VEL
LIN {X 0,Y 162.613,Z 411.302,A -85,B 0,C 180,E1 -24178.034,E2 -24178.034} C_VEL
LIN {X 0,Y 160.443,Z 420.323,A -85,B 0,C 180,E1 -24179.753,E2 -24179.753} C_VEL
LIN {X 0,Y 157.772,Z 431.307,A -85,B 0,C 180,E1 -24182.475,E2 -24182.475} C_VEL
LIN {X 0,Y 154.989,Z 441.031,A -85,B 0,C 180,E1 -24185.523,E2 -24185.523} C_VEL
LIN {X 0,Y 153.39,Z 446.912,A -85,B 0,C 180,E1 -24187.791,E2 -24187.791} C_VEL
LIN {X 0,Y 151.922,Z 452.129,A -85,B 0,C 180,E1 -24190.137,E2 -24190.137} C_VEL
LIN {X 0,Y 150.283,Z 455.615,A -85,B 0,C 180,E1 -24191.84,E2 -24191.84} C_VEL
LIN {X 0,Y 146.129,Z 460.734,A -85,B 0,C 180,E1 -24194.708,E2 -24194.708} C_VEL
LIN {X 0,Y 142.257,Z 465.132,A -85,B 0,C 180,E1 -24197.9,E2 -24197.9} C_VEL
LIN {X 0,Y 141.107,Z 467.487,A -85,B 0,C 180,E1 -24200.05,E2 -24200.05} C_VEL
LIN {X 0,Y 140.585,Z 471.369,A -85,B 0,C 180,E1 -24204.263,E2 -24204.263} C_VEL
LIN {X 0,Y 140.505,Z 473.4,A -85,B 0,C 180,E1 -24207.134,E2 -24207.134} C_VEL
LIN {X 0,Y 140.555,Z 475.005,A -85,B 0,C 180,E1 -24210.001,E2 -24210.001} C_VEL
LIN {X 0,Y 140.505,Z 476.196,A -85,B 0,C 180,E1 -24212.868,E2 -24212.868} C_VEL
LIN {X 0,Y 141.027,Z 477.319,A -85,B 0,C 180,E1 -24218.599,E2 -24218.599} C_VEL
LIN {X 0,Y 142.601,Z 476.913,A -85,B 0,C 180,E1 -24224.267,E2 -24224.267} C_VEL
LIN {X 0,Y 143.849,Z 476.136,A -85,B 0,C 180,E1 -24227.047,E2 -24227.047} C_VEL
LIN {X 0,Y 145.369,Z 474.936,A -85,B 0,C 180,E1 -24229.782,E2 -24229.782} C_VEL
LIN {X 0,Y 149.634,Z 471.35,A -85,B 0,C 180,E1 -24235.007,E2 -24235.007} C_VEL
LIN {X 0,Y 153.547,Z 467.499,A -85,B 0,C 180,E1 -24238.725,E2 -24238.725} C_VEL
LIN {X 0,Y 158.338,Z 462.199,A -85,B 0,C 180,E1 -24242.489,E2 -24242.489} C_VEL
LIN {X 0,Y 163.982,Z 455.204,A -85,B 0,C 180,E1 -24246.108,E2 -24246.108} C_VEL
LIN {X 0,Y 169.805,Z 447.22,A -85,B 0,C 180,E1 -24249.138,E2 -24249.138} C_VEL
LIN {X 0,Y 175.003,Z 439.099,A -85,B 0,C 180,E1 -24251.501,E2 -24251.501} C_VEL
LIN {X 0,Y 180.455,Z 429.228,A -85,B 0,C 180,E1 -24253.733,E2 -24253.733} C_VEL
LIN {X 0,Y 185.706,Z 418.078,A -85,B 0,C 180,E1 -24255.588,E2 -24255.588} C_VEL
LIN {X 0,Y 189.906,Z 407.207,A -85,B 0,C 180,E1 -24256.963,E2 -24256.963} C_VEL
LIN {X 0,Y 193.799,Z 394.414,A -85,B 0,C 180,E1 -24258.164,E2 -24258.164} C_VEL
LIN {X 0,Y 196.666,Z 381.232,A -85,B 0,C 180,E1 -24259.006,E2 -24259.006} C_VEL
LIN {X 0,Y 198.484,Z 367.301,A -85,B 0,C 180,E1 -24259.594,E2 -24259.594} C_VEL
LIN {X 0,Y 200.082,Z 347.44,A -85,B 0,C 180,E1 -24260.215,E2 -24260.215} C_VEL
LIN {X 0,Y 196.484,Z 338.733,A -85,B 0,C 180,E1 -24262.54,E2 -24262.54} C_VEL
LIN {X 0,Y 192.466,Z 330.212,A -85,B 0,C 180,E1 -24265.366,E2 -24265.366} C_VEL
LIN {X 0,Y 188.88,Z 323.323,A -85,B 0,C 180,E1 -24268.266,E2 -24268.266} C_VEL
LIN {X 0,Y 186.749,Z 319.376,A -85,B 0,C 180,E1 -24270.206,E2 -24270.206} C_VEL
LIN {X 0,Y 184.113,Z 314.925,A -85,B 0,C 180,E1 -24272.885,E2 -24272.885} C_VEL
LIN {X 0,Y 181.318,Z 310.353,A -85,B 0,C 180,E1 -24276.279,E2 -24276.279} C_VEL
LIN {X 0,Y 179.05,Z 307.613,A -85,B 0,C 180,E1 -24279.703,E2 -24279.703} C_VEL
LIN {X 0,Y 178.052,Z 305.481,A -85,B 0,C 180,E1 -24281.88,E2 -24281.88} C_VEL
LIN {X 0,Y 175.87,Z 303.37,A -85,B 0,C 180,E1 -24290.792,E2 -24290.792} C_VEL
LIN {X 0,Y 177.222,Z 304.473,A -85,B 0,C 180,E1 -24298.285,E2 -24298.285} C_VEL
LIN {X 0,Y 178.374,Z 305.485,A -85,B 0,C 180,E1 -24300.951,E2 -24300.951} C_VEL
LIN {X 0,Y 180.433,Z 309.203,A -85,B 0,C 180,E1 -24304.746,E2 -24304.746} C_VEL
LIN {X 0,Y 181.706,Z 310.513,A -85,B 0,C 180,E1 -24306.409,E2 -24306.409} C_VEL
LIN {X 0,Y 184.124,Z 314.292,A -85,B 0,C 180,E1 -24309.284,E2 -24309.284} C_VEL
LIN {X 0,Y 185.303,Z 316.006,A -85,B 0,C 180,E1 -24310.505,E2 -24310.505} C_VEL
LIN {X 0,Y 187.845,Z 319.8,A -85,B 0,C 180,E1 -24312.89,E2 -24312.89} C_VEL
LIN {X 0,Y 190.408,Z 323.938,A -85,B 0,C 180,E1 -24315.047,E2 -24315.047} C_VEL
LIN {X 0,Y 194.567,Z 331.853,A -85,B 0,C 180,E1 -24318.175,E2 -24318.175} C_VEL
LIN {X 0,Y 199.152,Z 341.64,A -85,B 0,C 180,E1 -24321.195,E2 -24321.195} C_VEL
LIN {X 0,Y 200.367,Z 344.667,A -85,B 0,C 180,E1 -24321.96,E2 -24321.96} C_VEL
LIN {X 0,Y 197.951,Z 371.25,A -85,B 0,C 180,E1 -24322.797,E2 -24322.797} C_VEL
LIN {X 0,Y 195.541,Z 384.932,A -85,B 0,C 180,E1 -24323.505,E2 -24323.505} C_VEL
LIN {X 0,Y 192.54,Z 396.882,A -85,B 0,C 180,E1 -24324.458,E2 -24324.458} C_VEL
LIN {X 0,Y 188.369,Z 409.288,A -85,B 0,C 180,E1 -24325.828,E2 -24325.828} C_VEL
LIN {X 0,Y 183.368,Z 421.222,A -85,B 0,C 180,E1 -24327.619,E2 -24327.619} C_VEL
LIN {X 0,Y 178.005,Z 431.636,A -85,B 0,C 180,E1 -24329.702,E2 -24329.702} C_VEL
LIN {X 0,Y 172.002,Z 441.692,A -85,B 0,C 180,E1 -24332.404,E2 -24332.404} C_VEL
LIN {X 0,Y 166.062,Z 450.165,A -85,B 0,C 180,E1 -24335.442,E2 -24335.442} C_VEL
LIN {X 0,Y 160.323,Z 457.329,A -85,B 0,C 180,E1 -24338.912,E2 -24338.912} C_VEL
LIN {X 0,Y 154.975,Z 463.26,A -85,B 0,C 180,E1 -24342.844,E2 -24342.844} C_VEL
LIN {X 0,Y 150.147,Z 467.896,A -85,B 0,C 180,E1 -24347.256,E2 -24347.256} C_VEL
LIN {X 0,Y 146.661,Z 470.844,A -85,B 0,C 180,E1 -24351.466,E2 -24351.466} C_VEL
LIN {X 0,Y 143.674,Z 472.828,A -85,B 0,C 180,E1 -24356.234,E2 -24356.234} C_VEL
LIN {X 0,Y 141.92,Z 473.559,A -85,B 0,C 180,E1 -24360.316,E2 -24360.316} C_VEL
LIN {X 0,Y 140.931,Z 473.528,A -85,B 0,C 180,E1 -24363.814,E2 -24363.814} C_VEL
LIN {X 0,Y 140.427,Z 473.136,A -85,B 0,C 180,E1 -24366.397,E2 -24366.397} C_VEL
LIN {X 0,Y 140.071,Z 472.246,A -85,B 0,C 180,E1 -24369.437,E2 -24369.437} C_VEL
LIN {X 0,Y 139.996,Z 470.911,A -85,B 0,C 180,E1 -24372.469,E2 -24372.469} C_VEL
LIN {X 0,Y 140.338,Z 468.072,A -85,B 0,C 180,E1 -24376.975,E2 -24376.975} C_VEL
LIN {X 0,Y 141.047,Z 464.169,A -85,B 0,C 180,E1 -24381.402,E2 -24381.402} C_VEL
LIN {X 0,Y 142.226,Z 459.104,A -85,B 0,C 180,E1 -24385.748,E2 -24385.748} C_VEL
LIN {X 0,Y 143.967,Z 452.73,A -85,B 0,C 180,E1 -24389.999,E2 -24389.999} C_VEL
LIN {X 0,Y 146.259,Z 444.747,A -85,B 0,C 180,E1 -24394.132,E2 -24394.132} C_VEL
LIN {X 0,Y 148.906,Z 435.826,A -85,B 0,C 180,E1 -24397.739,E2 -24397.739} C_VEL
LIN {X 0,Y 151.9,Z 425.491,A -85,B 0,C 180,E1 -24401.002,E2 -24401.002} C_VEL
LIN {X 0,Y 154.61,Z 415.352,A -85,B 0,C 180,E1 -24403.471,E2 -24403.471} C_VEL
LIN {X 0,Y 157.075,Z 404.354,A -85,B 0,C 180,E1 -24405.572,E2 -24405.572} C_VEL
LIN {X 0,Y 159.335,Z 392.212,A -85,B 0,C 180,E1 -24407.32,E2 -24407.32} C_VEL
LIN {X 0,Y 161.103,Z 379.734,A -85,B 0,C 180,E1 -24408.602,E2 -24408.602} C_VEL
LIN {X 0,Y 162.378,Z 366.75,A -85,B 0,C 180,E1 -24409.434,E2 -24409.434} C_VEL
LIN {X 0,Y 165.279,Z 314.237,A -85,B 0,C 180,E1 -24411.573,E2 -24411.573} C_VEL
LIN {X 0,Y 159.541,Z 298.162,A -85,B 0,C 180,E1 -24413.767,E2 -24413.767} C_VEL
LIN {X 0,Y 153.452,Z 286.715,A -85,B 0,C 180,E1 -24416.019,E2 -24416.019} C_VEL
LIN {X 0,Y 147.989,Z 277.546,A -85,B 0,C 180,E1 -24418.192,E2 -24418.192} C_VEL
LIN {X 0,Y 144.957,Z 273.003,A -85,B 0,C 180,E1 -24419.464,E2 -24419.464} C_VEL
LIN {X 0,Y 143.459,Z 270.405,A -85,B 0,C 180,E1 -24420.174,E2 -24420.174} C_VEL
LIN {X 0,Y 143.184,Z 269.361,A -85,B 0,C 180,E1 -24420.716,E2 -24420.716} C_VEL
LIN {X 0,Y 143.17,Z 269.138,A -85,B 0,C 180,E1 -24423.463,E2 -24423.463} C_VEL
LIN {X 0,Y 143.143,Z 269.142,A -85,B 0,C 180,E1 -24429.661,E2 -24429.661} C_VEL
LIN {X 0,Y 143.156,Z 269.123,A -85,B 0,C 180,E1 -24433.416,E2 -24433.416} C_VEL
LIN {X 0,Y 143.145,Z 269.15,A -85,B 0,C 180,E1 -24437.429,E2 -24437.429} C_VEL
LIN {X 0,Y 143.119,Z 269.113,A -85,B 0,C 180,E1 -24441.783,E2 -24441.783} C_VEL
LIN {X 0,Y 143.165,Z 269.15,A -85,B 0,C 180,E1 -24447.334,E2 -24447.334} C_VEL
LIN {X 0,Y 143.172,Z 269.095,A -85,B 0,C 180,E1 -24452.075,E2 -24452.075} C_VEL
LIN {X 0,Y 143.297,Z 269.135,A -85,B 0,C 180,E1 -24458.723,E2 -24458.723} C_VEL
LIN {X 0,Y 143.309,Z 269.079,A -85,B 0,C 180,E1 -24462.902,E2 -24462.902} C_VEL
LIN {X 0,Y 143.586,Z 269.075,A -85,B 0,C 180,E1 -24468.723,E2 -24468.723} C_VEL
LIN {X 0,Y 143.668,Z 269.088,A -85,B 0,C 180,E1 -24471.574,E2 -24471.574} C_VEL
LIN {X 0,Y 144.172,Z 268.975,A -85,B 0,C 180,E1 -24480.013,E2 -24480.013} C_VEL
LIN {X 0,Y 143.611,Z 269.049,A -85,B 0,C 180,E1 -24488.455,E2 -24488.455} C_VEL
LIN {X 0,Y 143.508,Z 269.059,A -85,B 0,C 180,E1 -24491.639,E2 -24491.639} C_VEL
LIN {X 0,Y 143.302,Z 269.128,A -85,B 0,C 180,E1 -24497.126,E2 -24497.126} C_VEL
LIN {X 0,Y 143.283,Z 269.095,A -85,B 0,C 180,E1 -24501.263,E2 -24501.263} C_VEL
LIN {X 0,Y 143.195,Z 269.128,A -85,B 0,C 180,E1 -24507.943,E2 -24507.943} C_VEL
LIN {X 0,Y 143.172,Z 269.155,A -85,B 0,C 180,E1 -24513.439,E2 -24513.439} C_VEL
LIN {X 0,Y 143.068,Z 269.16,A -85,B 0,C 180,E1 -24519.702,E2 -24519.702} C_VEL
LIN {X 0,Y 143.144,Z 269.405,A -85,B 0,C 180,E1 -24521.141,E2 -24521.141} C_VEL
LIN {X 0,Y 143.394,Z 270.425,A -85,B 0,C 180,E1 -24521.63,E2 -24521.63} C_VEL
LIN {X 0,Y 144.916,Z 273.099,A -85,B 0,C 180,E1 -24522.359,E2 -24522.359} C_VEL
LIN {X 0,Y 145.918,Z 274.401,A -85,B 0,C 180,E1 -24522.775,E2 -24522.775} C_VEL
LIN {X 0,Y 152.807,Z 285.749,A -85,B 0,C 180,E1 -24525.576,E2 -24525.576} C_VEL
LIN {X 0,Y 157.583,Z 296.172,A -85,B 0,C 180,E1 -24527.463,E2 -24527.463} C_VEL
LIN {X 0,Y 163.503,Z 312.502,A -85,B 0,C 180,E1 -24529.775,E2 -24529.775} C_VEL
LIN {X 0,Y 164.378,Z 315.684,A -85,B 0,C 180,E1 -24530.137,E2 -24530.137} C_VEL
LIN {X 0,Y 165.034,Z 323.625,A -85,B 0,C 180,E1 -24530.697,E2 -24530.697} C_VEL
LIN {X 0,Y 162.19,Z 373.534,A -85,B 0,C 180,E1 -24532.751,E2 -24532.751} C_VEL
LIN {X 0,Y 160.626,Z 386.725,A -85,B 0,C 180,E1 -24533.699,E2 -24533.699} C_VEL
LIN {X 0,Y 158.777,Z 398.968,A -85,B 0,C 180,E1 -24535.066,E2 -24535.066} C_VEL
LIN {X 0,Y 156.205,Z 411.258,A -85,B 0,C 180,E1 -24536.94,E2 -24536.94} C_VEL
LIN {X 0,Y 153.949,Z 420.272,A -85,B 0,C 180,E1 -24538.717,E2 -24538.717} C_VEL
LIN {X 0,Y 151.148,Z 431.247,A -85,B 0,C 180,E1 -24541.538,E2 -24541.538} C_VEL
LIN {X 0,Y 148.2,Z 441.054,A -85,B 0,C 180,E1 -24544.736,E2 -24544.736} C_VEL
LIN {X 0,Y 146.308,Z 447.592,A -85,B 0,C 180,E1 -24547.402,E2 -24547.402} C_VEL
LIN {X 0,Y 143.905,Z 455.736,A -85,B 0,C 180,E1 -24551.493,E2 -24551.493} C_VEL
LIN {X 0,Y 142.204,Z 462.254,A -85,B 0,C 180,E1 -24555.694,E2 -24555.694} C_VEL
LIN {X 0,Y 141.107,Z 467.487,A -85,B 0,C 180,E1 -24560.05,E2 -24560.05} C_VEL
LIN {X 0,Y 140.092,Z 469.65,A -85,B 0,C 180,E1 -24562.263,E2 -24562.263} C_VEL
LIN {X 0,Y 136.948,Z 472.537,A -85,B 0,C 180,E1 -24565.969,E2 -24565.969} C_VEL
LIN {X 0,Y 134.475,Z 474.336,A -85,B 0,C 180,E1 -24569.098,E2 -24569.098} C_VEL
LIN {X 0,Y 133.467,Z 475.435,A -85,B 0,C 180,E1 -24571.573,E2 -24571.573} C_VEL
LIN {X 0,Y 133.401,Z 475.715,A -85,B 0,C 180,E1 -24572.414,E2 -24572.414} C_VEL
LIN {X 0,Y 133.545,Z 476.793,A -85,B 0,C 180,E1 -24576.043,E2 -24576.043} C_VEL
LIN {X 0,Y 134.002,Z 477.2,A -85,B 0,C 180,E1 -24579.054,E2 -24579.054} C_VEL
LIN {X 0,Y 135.701,Z 476.876,A -85,B 0,C 180,E1 -24585.009,E2 -24585.009} C_VEL
LIN {X 0,Y 137.041,Z 476.155,A -85,B 0,C 180,E1 -24587.922,E2 -24587.922} C_VEL
LIN {X 0,Y 138.69,Z 475.029,A -85,B 0,C 180,E1 -24590.777,E2 -24590.777} C_VEL
LIN {X 0,Y 143.245,Z 471.532,A -85,B 0,C 180,E1 -24596.205,E2 -24596.205} C_VEL
LIN {X 0,Y 147.358,Z 467.776,A -85,B 0,C 180,E1 -24600.052,E2 -24600.052} C_VEL
LIN {X 0,Y 152.061,Z 462.939,A -85,B 0,C 180,E1 -24603.685,E2 -24603.685} C_VEL
LIN {X 0,Y 157.367,Z 456.874,A -85,B 0,C 180,E1 -24607.079,E2 -24607.079} C_VEL
LIN {X 0,Y 163.323,Z 449.352,A -85,B 0,C 180,E1 -24610.202,E2 -24610.202} C_VEL
LIN {X 0,Y 169.802,Z 439.928,A -85,B 0,C 180,E1 -24613.073,E2 -24613.073} C_VEL
LIN {X 0,Y 175.448,Z 430.244,A -85,B 0,C 180,E1 -24615.319,E2 -24615.319} C_VEL
LIN {X 0,Y 180.862,Z 419.455,A -85,B 0,C 180,E1 -24617.177,E2 -24617.177} C_VEL
LIN {X 0,Y 185.195,Z 408.935,A -85,B 0,C 180,E1 -24618.548,E2 -24618.548} C_VEL
LIN {X 0,Y 189.307,Z 396.34,A -85,B 0,C 180,E1 -24619.764,E2 -24619.764} C_VEL
LIN {X 0,Y 192.439,Z 383.261,A -85,B 0,C 180,E1 -24620.661,E2 -24620.661} C_VEL
LIN {X 0,Y 194.472,Z 369.673,A -85,B 0,C 180,E1 -24621.255,E2 -24621.255} C_VEL
LIN {X 0,Y 196.111,Z 350.213,A -85,B 0,C 180,E1 -24621.889,E2 -24621.889} C_VEL
LIN {X 0,Y 191.984,Z 340.328,A -85,B 0,C 180,E1 -24624.816,E2 -24624.816} C_VEL
LIN {X 0,Y 188.547,Z 332.971,A -85,B 0,C 180,E1 -24627.584,E2 -24627.584} C_VEL
LIN {X 0,Y 185.186,Z 326.203,A -85,B 0,C 180,E1 -24630.7,E2 -24630.7} C_VEL
LIN {X 0,Y 182.49,Z 321.478,A -85,B 0,C 180,E1 -24633.57,E2 -24633.57} C_VEL
LIN {X 0,Y 179.827,Z 317.048,A -85,B 0,C 180,E1 -24636.985,E2 -24636.985} C_VEL
LIN {X 0,Y 177.427,Z 313.571,A -85,B 0,C 180,E1 -24641.116,E2 -24641.116} C_VEL
LIN {X 0,Y 176.851,Z 312.384,A -85,B 0,C 180,E1 -24642.509,E2 -24642.509} C_VEL
LIN {X 0,Y 174.981,Z 310.406,A -85,B 0,C 180,E1 -24650.745,E2 -24650.745} C_VEL
LIN {X 0,Y 176.539,Z 311.674,A -85,B 0,C 180,E1 -24658.849,E2 -24658.849} C_VEL
LIN {X 0,Y 177.226,Z 312.399,A -85,B 0,C 180,E1 -24660.471,E2 -24660.471} C_VEL
LIN {X 0,Y 179.146,Z 315.995,A -85,B 0,C 180,E1 -24664.226,E2 -24664.226} C_VEL
LIN {X 0,Y 180.303,Z 317.313,A -85,B 0,C 180,E1 -24665.845,E2 -24665.845} C_VEL
LIN {X 0,Y 182.727,Z 321.105,A -85,B 0,C 180,E1 -24668.839,E2 -24668.839} C_VEL
LIN {X 0,Y 186.042,Z 326.379,A -85,B 0,C 180,E1 -24672.216,E2 -24672.216} C_VEL
LIN {X 0,Y 188.373,Z 330.302,A -85,B 0,C 180,E1 -24674.282,E2 -24674.282} C_VEL
LIN {X 0,Y 192.349,Z 338.342,A -85,B 0,C 180,E1 -24677.466,E2 -24677.466} C_VEL
LIN {X 0,Y 196.341,Z 347.462,A -85,B 0,C 180,E1 -24680.26,E2 -24680.26} C_VEL
LIN {X 0,Y 194.145,Z 371.34,A -85,B 0,C 180,E1 -24681.046,E2 -24681.046} C_VEL
LIN {X 0,Y 191.659,Z 385.076,A -85,B 0,C 180,E1 -24681.753,E2 -24681.753} C_VEL
LIN {X 0,Y 188.205,Z 398.085,A -85,B 0,C 180,E1 -24682.796,E2 -24682.796} C_VEL
LIN {X 0,Y 183.929,Z 410.164,A -85,B 0,C 180,E1 -24684.141,E2 -24684.141} C_VEL
LIN {X 0,Y 178.757,Z 421.909,A -85,B 0,C 180,E1 -24685.926,E2 -24685.926} C_VEL
LIN {X 0,Y 173.164,Z 432.269,A -85,B 0,C 180,E1 -24688.024,E2 -24688.024} C_VEL
LIN {X 0,Y 167.911,Z 440.703,A -85,B 0,C 180,E1 -24690.27,E2 -24690.27} C_VEL
LIN {X 0,Y 161.779,Z 449.27,A -85,B 0,C 180,E1 -24693.252,E2 -24693.252} C_VEL
LIN {X 0,Y 155.638,Z 456.632,A -85,B 0,C 180,E1 -24696.723,E2 -24696.723} C_VEL
LIN {X 0,Y 151.016,Z 461.586,A -85,B 0,C 180,E1 -24699.835,E2 -24699.835} C_VEL
LIN {X 0,Y 146.095,Z 466.261,A -85,B 0,C 180,E1 -24703.814,E2 -24703.814} C_VEL
LIN {X 0,Y 142.101,Z 469.609,A -85,B 0,C 180,E1 -24707.869,E2 -24707.869} C_VEL
LIN {X 0,Y 138.571,Z 472.084,A -85,B 0,C 180,E1 -24712.51,E2 -24712.51} C_VEL
LIN {X 0,Y 136.787,Z 473.074,A -85,B 0,C 180,E1 -24715.585,E2 -24715.585} C_VEL
LIN {X 0,Y 135.33,Z 473.628,A -85,B 0,C 180,E1 -24718.712,E2 -24718.712} C_VEL
LIN {X 0,Y 133.966,Z 473.625,A -85,B 0,C 180,E1 -24723.07,E2 -24723.07} C_VEL
LIN {X 0,Y 133.063,Z 472.567,A -85,B 0,C 180,E1 -24728.301,E2 -24728.301} C_VEL
LIN {X 0,Y 132.898,Z 471.021,A -85,B 0,C 180,E1 -24732.102,E2 -24732.102} C_VEL
LIN {X 0,Y 133.351,Z 467.491,A -85,B 0,C 180,E1 -24737.829,E2 -24737.829} C_VEL
LIN {X 0,Y 134.4,Z 462.422,A -85,B 0,C 180,E1 -24743.343,E2 -24743.343} C_VEL
LIN {X 0,Y 136.132,Z 455.956,A -85,B 0,C 180,E1 -24748.52,E2 -24748.52} C_VEL
LIN {X 0,Y 138.266,Z 448.758,A -85,B 0,C 180,E1 -24752.913,E2 -24752.913} C_VEL
LIN {X 0,Y 140.552,Z 441.252,A -85,B 0,C 180,E1 -24756.531,E2 -24756.531} C_VEL
LIN {X 0,Y 143.34,Z 432.261,A -85,B 0,C 180,E1 -24759.964,E2 -24759.964} C_VEL
LIN {X 0,Y 146.548,Z 421.479,A -85,B 0,C 180,E1 -24763.166,E2 -24763.166} C_VEL
LIN {X 0,Y 149.447,Z 410.354,A -85,B 0,C 180,E1 -24765.687,E2 -24765.687} C_VEL
LIN {X 0,Y 152.141,Z 397.895,A -85,B 0,C 180,E1 -24767.819,E2 -24767.819} C_VEL
LIN {X 0,Y 154.125,Z 386.108,A -85,B 0,C 180,E1 -24769.304,E2 -24769.304} C_VEL
LIN {X 0,Y 155.752,Z 373.313,A -85,B 0,C 180,E1 -24770.382,E2 -24770.382} C_VEL
LIN {X 0,Y 156.998,Z 355.677,A -85,B 0,C 180,E1 -24771.237,E2 -24771.237} C_VEL
LIN {X 0,Y 159.291,Z 315.931,A -85,B 0,C 180,E1 -24772.858,E2 -24772.858} C_VEL
LIN {X 0,Y 154.123,Z 301.368,A -85,B 0,C 180,E1 -24774.983,E2 -24774.983} C_VEL
LIN {X 0,Y 147.025,Z 288.099,A -85,B 0,C 180,E1 -24777.831,E2 -24777.831} C_VEL
LIN {X 0,Y 142.576,Z 280.961,A -85,B 0,C 180,E1 -24779.748,E2 -24779.748} C_VEL
LIN {X 0,Y 140.671,Z 277.921,A -85,B 0,C 180,E1 -24780.623,E2 -24780.623} C_VEL
LIN {X 0,Y 138.462,Z 274.487,A -85,B 0,C 180,E1 -24781.67,E2 -24781.67} C_VEL
LIN {X 0,Y 136.719,Z 272.062,A -85,B 0,C 180,E1 -24782.515,E2 -24782.515} C_VEL
LIN {X 0,Y 136.224,Z 270.474,A -85,B 0,C 180,E1 -24783.093,E2 -24783.093} C_VEL
LIN {X 0,Y 136.079,Z 270.015,A -85,B 0,C 180,E1 -24784.303,E2 -24784.303} C_VEL
LIN {X 0,Y 136.107,Z 270.023,A -85,B 0,C 180,E1 -24789.261,E2 -24789.261} C_VEL
LIN {X 0,Y 136.09,Z 270.004,A -85,B 0,C 180,E1 -24793.72,E2 -24793.72} C_VEL
LIN {X 0,Y 136.091,Z 270.021,A -85,B 0,C 180,E1 -24797.85,E2 -24797.85} C_VEL
LIN {X 0,Y 136.071,Z 269.99,A -85,B 0,C 180,E1 -24801.718,E2 -24801.718} C_VEL
LIN {X 0,Y 136.071,Z 270.032,A -85,B 0,C 180,E1 -24805.728,E2 -24805.728} C_VEL
LIN {X 0,Y 136.128,Z 269.971,A -85,B 0,C 180,E1 -24812.329,E2 -24812.329} C_VEL
LIN {X 0,Y 136.264,Z 270.01,A -85,B 0,C 180,E1 -24818.851,E2 -24818.851} C_VEL
LIN {X 0,Y 136.27,Z 269.945,A -85,B 0,C 180,E1 -24825.071,E2 -24825.071} C_VEL
LIN {X 0,Y 136.488,Z 269.946,A -85,B 0,C 180,E1 -24828.128,E2 -24828.128} C_VEL
LIN {X 0,Y 136.592,Z 269.97,A -85,B 0,C 180,E1 -24831.134,E2 -24831.134} C_VEL
LIN {X 0,Y 137.129,Z 269.851,A -85,B 0,C 180,E1 -24840.013,E2 -24840.013} C_VEL
LIN {X 0,Y 136.54,Z 269.925,A -85,B 0,C 180,E1 -24848.896,E2 -24848.896} C_VEL
LIN {X 0,Y 136.445,Z 269.94,A -85,B 0,C 180,E1 -24851.903,E2 -24851.903} C_VEL
LIN {X 0,Y 136.216,Z 269.995,A -85,B 0,C 180,E1 -24858.046,E2 -24858.046} C_VEL
LIN {X 0,Y 136.204,Z 269.977,A -85,B 0,C 180,E1 -24861.758,E2 -24861.758} C_VEL
LIN {X 0,Y 136.105,Z 270.005,A -85,B 0,C 180,E1 -24868.622,E2 -24868.622} C_VEL
LIN {X 0,Y 136.082,Z 270.03,A -85,B 0,C 180,E1 -24874.632,E2 -24874.632} C_VEL
LIN {X 0,Y 136.072,Z 270.244,A -85,B 0,C 180,E1 -24878.47,E2 -24878.47} C_VEL
LIN {X 0,Y 136.29,Z 271.242,A -85,B 0,C 180,E1 -24879.059,E2 -24879.059} C_VEL
LIN {X 0,Y 137.871,Z 273.992,A -85,B 0,C 180,E1 -24879.908,E2 -24879.908} C_VEL
LIN {X 0,Y 138.993,Z 275.202,A -85,B 0,C 180,E1 -24880.412,E2 -24880.412} C_VEL
LIN {X 0,Y 141.153,Z 278.655,A -85,B 0,C 180,E1 -24881.431,E2 -24881.431} C_VEL
LIN {X 0,Y 148.052,Z 290.091,A -85,B 0,C 180,E1 -24884.441,E2 -24884.441} C_VEL
LIN {X 0,Y 152.558,Z 300.278,A -85,B 0,C 180,E1 -24886.361,E2 -24886.361} C_VEL
LIN {X 0,Y 158.109,Z 316.135,A -85,B 0,C 180,E1 -24888.702,E2 -24888.702} C_VEL
LIN {X 0,Y 158.753,Z 320.031,A -85,B 0,C 180,E1 -24889.071,E2 -24889.071} C_VEL
LIN {X 0,Y 158.936,Z 325.734,A -85,B 0,C 180,E1 -24889.424,E2 -24889.424} C_VEL
LIN {X 0,Y 156.105,Z 373.597,A -85,B 0,C 180,E1 -24891.447,E2 -24891.447} C_VEL
LIN {X 0,Y 154.477,Z 386.733,A -85,B 0,C 180,E1 -24892.417,E2 -24892.417} C_VEL
LIN {X 0,Y 152.544,Z 398.948,A -85,B 0,C 180,E1 -24893.823,E2 -24893.823} C_VEL
LIN {X 0,Y 149.86,Z 411.214,A -85,B 0,C 180,E1 -24895.754,E2 -24895.754} C_VEL
LIN {X 0,Y 147.51,Z 420.221,A -85,B 0,C 180,E1 -24897.59,E2 -24897.59} C_VEL
LIN {X 0,Y 144.563,Z 431.186,A -85,B 0,C 180,E1 -24900.514,E2 -24900.514} C_VEL
LIN {X 0,Y 141.732,Z 440.081,A -85,B 0,C 180,E1 -24903.496,E2 -24903.496} C_VEL
LIN {X 0,Y 139.754,Z 446.77,A -85,B 0,C 180,E1 -24906.279,E2 -24906.279} C_VEL
LIN {X 0,Y 137.168,Z 455.039,A -85,B 0,C 180,E1 -24910.548,E2 -24910.548} C_VEL
LIN {X 0,Y 135.315,Z 461.677,A -85,B 0,C 180,E1 -24914.949,E2 -24914.949} C_VEL
LIN {X 0,Y 134.037,Z 467.336,A -85,B 0,C 180,E1 -24919.844,E2 -24919.844} C_VEL
LIN {X 0,Y 133.531,Z 470.997,A -85,B 0,C 180,E1 -24923.959,E2 -24923.959} C_VEL
LIN {X 0,Y 133.419,Z 473.085,A -85,B 0,C 180,E1 -24926.982,E2 -24926.982} C_VEL
LIN {X 0,Y 133.475,Z 474.732,A -85,B 0,C 180,E1 -24930.001,E2 -24930.001} C_VEL
LIN {X 0,Y 133.401,Z 475.715,A -85,B 0,C 180,E1 -24932.414,E2 -24932.414} C_VEL
LIN {X 0,Y 132.842,Z 476.574,A -85,B 0,C 180,E1 -24934.917,E2 -24934.917} C_VEL
LIN {X 0,Y 130.474,Z 477.306,A -85,B 0,C 180,E1 -24939.099,E2 -24939.099} C_VEL
LIN {X 0,Y 128.832,Z 477.298,A -85,B 0,C 180,E1 -24942.558,E2 -24942.558} C_VEL
LIN {X 0,Y 128.662,Z 476.961,A -85,B 0,C 180,E1 -24945.202,E2 -24945.202} C_VEL
LIN {X 0,Y 128.927,Z 476.787,A -85,B 0,C 180,E1 -24946.073,E2 -24946.073} C_VEL
LIN {X 0,Y 132.063,Z 475.106,A -85,B 0,C 180,E1 -24951.872,E2 -24951.872} C_VEL
LIN {X 0,Y 134.313,Z 473.619,A -85,B 0,C 180,E1 -24954.748,E2 -24954.748} C_VEL
LIN {X 0,Y 138.305,Z 470.627,A -85,B 0,C 180,E1 -24958.866,E2 -24958.866} C_VEL
LIN {X 0,Y 142.879,Z 466.621,A -85,B 0,C 180,E1 -24962.758,E2 -24962.758} C_VEL
LIN {X 0,Y 147.987,Z 461.5,A -85,B 0,C 180,E1 -24966.416,E2 -24966.416} C_VEL
LIN {X 0,Y 153.81,Z 455.077,A -85,B 0,C 180,E1 -24969.77,E2 -24969.77} C_VEL
LIN {X 0,Y 160.25,Z 447.099,A -85,B 0,C 180,E1 -24972.827,E2 -24972.827} C_VEL
LIN {X 0,Y 165.9,Z 438.993,A -85,B 0,C 180,E1 -24975.202,E2 -24975.202} C_VEL
LIN {X 0,Y 171.776,Z 429.146,A -85,B 0,C 180,E1 -24977.43,E2 -24977.43} C_VEL
LIN {X 0,Y 177.424,Z 418.025,A -85,B 0,C 180,E1 -24979.251,E2 -24979.251} C_VEL
LIN {X 0,Y 181.924,Z 407.181,A -85,B 0,C 180,E1 -24980.591,E2 -24980.591} C_VEL
LIN {X 0,Y 185.849,Z 395.239,A -85,B 0,C 180,E1 -24981.691,E2 -24981.691} C_VEL
LIN {X 0,Y 188.88,Z 382.653,A -85,B 0,C 180,E1 -24982.517,E2 -24982.517} C_VEL
LIN {X 0,Y 190.923,Z 369.093,A -85,B 0,C 180,E1 -24983.098,E2 -24983.098} C_VEL
LIN {X 0,Y 192.3,Z 353.268,A -85,B 0,C 180,E1 -24983.616,E2 -24983.616} C_VEL
LIN {X 0,Y 188.557,Z 343.897,A -85,B 0,C 180,E1 -24986.581,E2 -24986.581} C_VEL
LIN {X 0,Y 185.238,Z 336.538,A -85,B 0,C 180,E1 -24989.575,E2 -24989.575} C_VEL
LIN {X 0,Y 182.594,Z 331.282,A -85,B 0,C 180,E1 -24992.285,E2 -24992.285} C_VEL
LIN {X 0,Y 180.586,Z 327.523,A -85,B 0,C 180,E1 -24994.644,E2 -24994.644} C_VEL
LIN {X 0,Y 178.566,Z 323.903,A -85,B 0,C 180,E1 -24997.425,E2 -24997.425} C_VEL
LIN {X 0,Y 176.243,Z 320.354,A -85,B 0,C 180,E1 -25001.688,E2 -25001.688} C_VEL
LIN {X 0,Y 175.785,Z 319.325,A -85,B 0,C 180,E1 -25002.883,E2 -25002.883} C_VEL
LIN {X 0,Y 174.088,Z 317.468,A -85,B 0,C 180,E1 -25010.697,E2 -25010.697} C_VEL
LIN {X 0,Y 175.414,Z 318.581,A -85,B 0,C 180,E1 -25018.268,E2 -25018.268} C_VEL
LIN {X 0,Y 176.096,Z 319.288,A -85,B 0,C 180,E1 -25019.99,E2 -25019.99} C_VEL
LIN {X 0,Y 178.062,Z 322.975,A -85,B 0,C 180,E1 -25023.987,E2 -25023.987} C_VEL
LIN {X 0,Y 179.034,Z 324.337,A -85,B 0,C 180,E1 -25025.445,E2 -25025.445} C_VEL
LIN {X 0,Y 181.759,Z 328.734,A -85,B 0,C 180,E1 -25028.887,E2 -25028.887} C_VEL
LIN {X 0,Y 184.409,Z 333.187,A -85,B 0,C 180,E1 -25031.669,E2 -25031.669} C_VEL
LIN {X 0,Y 186.352,Z 336.655,A -85,B 0,C 180,E1 -25033.484,E2 -25033.484} C_VEL
LIN {X 0,Y 189.749,Z 343.905,A -85,B 0,C 180,E1 -25036.399,E2 -25036.399} C_VEL
LIN {X 0,Y 192.564,Z 350.623,A -85,B 0,C 180,E1 -25038.555,E2 -25038.555} C_VEL
LIN {X 0,Y 190.353,Z 372.684,A -85,B 0,C 180,E1 -25039.285,E2 -25039.285} C_VEL
LIN {X 0,Y 187.826,Z 385.789,A -85,B 0,C 180,E1 -25039.958,E2 -25039.958} C_VEL
LIN {X 0,Y 184.385,Z 398.238,A -85,B 0,C 180,E1 -25040.958,E2 -25040.958} C_VEL
LIN {X 0,Y 180.268,Z 409.563,A -85,B 0,C 180,E1 -25042.192,E2 -25042.192} C_VEL
LIN {X 0,Y 174.943,Z 421.4,A -85,B 0,C 180,E1 -25043.943,E2 -25043.943} C_VEL
LIN {X 0,Y 169.097,Z 431.864,A -85,B 0,C 180,E1 -25046.001,E2 -25046.001} C_VEL
LIN {X 0,Y 163.855,Z 440.04,A -85,B 0,C 180,E1 -25048.138,E2 -25048.138} C_VEL
LIN {X 0,Y 157.739,Z 448.301,A -85,B 0,C 180,E1 -25050.942,E2 -25050.942} C_VEL
LIN {X 0,Y 151.211,Z 455.93,A -85,B 0,C 180,E1 -25054.412,E2 -25054.412} C_VEL
LIN {X 0,Y 146.26,Z 461.016,A -85,B 0,C 180,E1 -25057.546,E2 -25057.546} C_VEL
LIN {X 0,Y 140.904,Z 465.867,A -85,B 0,C 180,E1 -25061.567,E2 -25061.567} C_VEL
LIN {X 0,Y 135.89,Z 469.775,A -85,B 0,C 180,E1 -25066.368,E2 -25066.368} C_VEL
LIN {X 0,Y 132.586,Z 471.965,A -85,B 0,C 180,E1 -25070.498,E2 -25070.498} C_VEL
LIN {X 0,Y 130.4,Z 473.08,A -85,B 0,C 180,E1 -25073.916,E2 -25073.916} C_VEL
LIN {X 0,Y 128.874,Z 473.649,A -85,B 0,C 180,E1 -25076.951,E2 -25076.951} C_VEL
LIN {X 0,Y 127.036,Z 473.721,A -85,B 0,C 180,E1 -25082.236,E2 -25082.236} C_VEL
LIN {X 0,Y 126.084,Z 472.83,A -85,B 0,C 180,E1 -25087.033,E2 -25087.033} C_VEL
LIN {X 0,Y 125.81,Z 471.119,A -85,B 0,C 180,E1 -25091.687,E2 -25091.687} C_VEL
LIN {X 0,Y 126.133,Z 468.008,A -85,B 0,C 180,E1 -25097.121,E2 -25097.121} C_VEL
LIN {X 0,Y 126.985,Z 463.869,A -85,B 0,C 180,E1 -25102.206,E2 -25102.206} C_VEL
LIN {X 0,Y 128.583,Z 457.864,A -85,B 0,C 180,E1 -25107.65,E2 -25107.65} C_VEL
LIN {X 0,Y 130.64,Z 451.101,A -85,B 0,C 180,E1 -25112.311,E2 -25112.311} C_VEL
LIN {X 0,Y 133.362,Z 442.705,A -85,B 0,C 180,E1 -25116.809,E2 -25116.809} C_VEL
LIN {X 0,Y 136.397,Z 433.325,A -85,B 0,C 180,E1 -25120.673,E2 -25120.673} C_VEL
LIN {X 0,Y 139.555,Z 423.352,A -85,B 0,C 180,E1 -25123.839,E2 -25123.839} C_VEL
LIN {X 0,Y 142.565,Z 412.712,A -85,B 0,C 180,E1 -25126.466,E2 -25126.466} C_VEL
LIN {X 0,Y 145.334,Z 400.967,A -85,B 0,C 180,E1 -25128.684,E2 -25128.684} C_VEL
LIN {X 0,Y 147.594,Z 388.774,A -85,B 0,C 180,E1 -25130.376,E2 -25130.376} C_VEL
LIN {X 0,Y 149.487,Z 375.456,A -85,B 0,C 180,E1 -25131.639,E2 -25131.639} C_VEL
LIN {X 0,Y 150.612,Z 361.992,A -85,B 0,C 180,E1 -25132.399,E2 -25132.399} C_VEL
LIN {X 0,Y 153.342,Z 317.534,A -85,B 0,C 180,E1 -25134.259,E2 -25134.259} C_VEL
LIN {X 0,Y 148.604,Z 304.2,A -85,B 0,C 180,E1 -25136.359,E2 -25136.359} C_VEL
LIN {X 0,Y 140.921,Z 289.927,A -85,B 0,C 180,E1 -25139.716,E2 -25139.716} C_VEL
LIN {X 0,Y 134.403,Z 279.659,A -85,B 0,C 180,E1 -25142.866,E2 -25142.866} C_VEL
LIN {X 0,Y 132.269,Z 276.322,A -85,B 0,C 180,E1 -25143.996,E2 -25143.996} C_VEL
LIN {X 0,Y 129.767,Z 273.351,A -85,B 0,C 180,E1 -25145.324,E2 -25145.324} C_VEL
LIN {X 0,Y 129.088,Z 271.527,A -85,B 0,C 180,E1 -25145.986,E2 -25145.986} C_VEL
LIN {X 0,Y 129.011,Z 270.948,A -85,B 0,C 180,E1 -25146.814,E2 -25146.814} C_VEL
LIN {X 0,Y 129.032,Z 270.885,A -85,B 0,C 180,E1 -25150.812,E2 -25150.812} C_VEL
LIN {X 0,Y 129.012,Z 270.898,A -85,B 0,C 180,E1 -25155.085,E2 -25155.085} C_VEL
LIN {X 0,Y 128.994,Z 270.878,A -85,B 0,C 180,E1 -25159.706,E2 -25159.706} C_VEL
LIN {X 0,Y 129.003,Z 270.897,A -85,B 0,C 180,E1 -25164.802,E2 -25164.802} C_VEL
LIN {X 0,Y 128.997,Z 270.865,A -85,B 0,C 180,E1 -25170.655,E2 -25170.655} C_VEL
LIN {X 0,Y 129.121,Z 270.899,A -85,B 0,C 180,E1 -25177.62,E2 -25177.62} C_VEL
LIN {X 0,Y 129.167,Z 270.865,A -85,B 0,C 180,E1 -25180.962,E2 -25180.962} C_VEL
LIN {X 0,Y 129.408,Z 270.821,A -85,B 0,C 180,E1 -25187.833,E2 -25187.833} C_VEL
LIN {X 0,Y 129.516,Z 270.85,A -85,B 0,C 180,E1 -25190.646,E2 -25190.646} C_VEL
LIN {X 0,Y 130.084,Z 270.727,A -85,B 0,C 180,E1 -25200.014,E2 -25200.014} C_VEL
LIN {X 0,Y 129.467,Z 270.802,A -85,B 0,C 180,E1 -25209.386,E2 -25209.386} C_VEL
LIN {X 0,Y 129.348,Z 270.829,A -85,B 0,C 180,E1 -25212.566,E2 -25212.566} C_VEL
LIN {X 0,Y 129.138,Z 270.864,A -85,B 0,C 180,E1 -25219.073,E2 -25219.073} C_VEL
LIN {X 0,Y 129.117,Z 270.863,A -85,B 0,C 180,E1 -25222.411,E2 -25222.411} C_VEL
LIN {X 0,Y 129.035,Z 270.915,A -85,B 0,C 180,E1 -25225.846,E2 -25225.846} C_VEL
LIN {X 0,Y 129.028,Z 270.883,A -85,B 0,C 180,E1 -25229.369,E2 -25229.369} C_VEL
LIN {X 0,Y 129.053,Z 271.157,A -85,B 0,C 180,E1 -25235.539,E2 -25235.539} C_VEL
LIN {X 0,Y 129.289,Z 272.141,A -85,B 0,C 180,E1 -25236.146,E2 -25236.146} C_VEL
LIN {X 0,Y 130.801,Z 274.808,A -85,B 0,C 180,E1 -25237.085,E2 -25237.085} C_VEL
LIN {X 0,Y 132.076,Z 276.195,A -85,B 0,C 180,E1 -25237.745,E2 -25237.745} C_VEL
LIN {X 0,Y 134.287,Z 279.645,A -85,B 0,C 180,E1 -25238.92,E2 -25238.92} C_VEL
LIN {X 0,Y 140.088,Z 288.761,A -85,B 0,C 180,E1 -25241.747,E2 -25241.747} C_VEL
LIN {X 0,Y 144.274,Z 296.358,A -85,B 0,C 180,E1 -25243.654,E2 -25243.654} C_VEL
LIN {X 0,Y 148.641,Z 307.253,A -85,B 0,C 180,E1 -25245.669,E2 -25245.669} C_VEL
LIN {X 0,Y 152.751,Z 319.668,A -85,B 0,C 180,E1 -25247.541,E2 -25247.541} C_VEL
LIN {X 0,Y 153.112,Z 324.689,A -85,B 0,C 180,E1 -25247.924,E2 -25247.924} C_VEL
LIN {X 0,Y 150.099,Z 373.382,A -85,B 0,C 180,E1 -25250.035,E2 -25250.035} C_VEL
LIN {X 0,Y 148.411,Z 386.557,A -85,B 0,C 180,E1 -25251.03,E2 -25251.03} C_VEL
LIN {X 0,Y 146.395,Z 398.802,A -85,B 0,C 180,E1 -25252.478,E2 -25252.478} C_VEL
LIN {X 0,Y 143.585,Z 411.082,A -85,B 0,C 180,E1 -25254.464,E2 -25254.464} C_VEL
LIN {X 0,Y 141.132,Z 420.094,A -85,B 0,C 180,E1 -25256.36,E2 -25256.36} C_VEL
LIN {X 0,Y 138.022,Z 431.068,A -85,B 0,C 180,E1 -25259.391,E2 -25259.391} C_VEL
LIN {X 0,Y 134.813,Z 440.879,A -85,B 0,C 180,E1 -25262.862,E2 -25262.862} C_VEL
LIN {X 0,Y 132.206,Z 448.92,A -85,B 0,C 180,E1 -25266.505,E2 -25266.505} C_VEL
LIN {X 0,Y 129.633,Z 456.737,A -85,B 0,C 180,E1 -25271.018,E2 -25271.018} C_VEL
LIN {X 0,Y 127.923,Z 462.993,A -85,B 0,C 180,E1 -25275.688,E2 -25275.688} C_VEL
LIN {X 0,Y 126.824,Z 467.931,A -85,B 0,C 180,E1 -25280.431,E2 -25280.431} C_VEL
LIN {X 0,Y 126.353,Z 471.712,A -85,B 0,C 180,E1 -25285.215,E2 -25285.215} C_VEL
LIN {X 0,Y 126.385,Z 474.447,A -85,B 0,C 180,E1 -25290.001,E2 -25290.001} C_VEL
LIN {X 0,Y 126.329,Z 475.716,A -85,B 0,C 180,E1 -25293.19,E2 -25293.19} C_VEL
LIN {X 0,Y 126.978,Z 477.078,A -85,B 0,C 180,E1 -25299.559,E2 -25299.559} C_VEL
LIN {X 0,Y 128.827,Z 476.84,A -85,B 0,C 180,E1 -25305.83,E2 -25305.83} C_VEL
LIN {X 0,Y 128.927,Z 476.787,A -85,B 0,C 180,E1 -25306.073,E2 -25306.073} C_VEL
LIN {X 0,Y 129.484,Z 476.26,A -85,B 0,C 180,E1 -25308.666,E2 -25308.666} C_VEL
LIN {X 0,Y 129.253,Z 474.891,A -85,B 0,C 180,E1 -25313.015,E2 -25313.015} C_VEL
LIN {X 0,Y 129.477,Z 473.369,A -85,B 0,C 180,E1 -25316.463,E2 -25316.463} C_VEL
LIN {X 0,Y 130.693,Z 471.91,A -85,B 0,C 180,E1 -25318.924,E2 -25318.924} C_VEL
LIN {X 0,Y 131.395,Z 471.343,A -85,B 0,C 180,E1 -25319.691,E2 -25319.691} C_VEL
LIN {X 0,Y 136.976,Z 466.912,A -85,B 0,C 180,E1 -25324.361,E2 -25324.361} C_VEL
LIN {X 0,Y 142.353,Z 461.9,A -85,B 0,C 180,E1 -25328.108,E2 -25328.108} C_VEL
LIN {X 0,Y 148.441,Z 455.62,A -85,B 0,C 180,E1 -25331.517,E2 -25331.517} C_VEL
LIN {X 0,Y 155.156,Z 447.776,A -85,B 0,C 180,E1 -25334.596,E2 -25334.596} C_VEL
LIN {X 0,Y 161.022,Z 439.822,A -85,B 0,C 180,E1 -25336.977,E2 -25336.977} C_VEL
LIN {X 0,Y 167.737,Z 429.102,A -85,B 0,C 180,E1 -25339.414,E2 -25339.414} C_VEL
LIN {X 0,Y 173.574,Z 417.998,A -85,B 0,C 180,E1 -25341.21,E2 -25341.21} C_VEL
LIN {X 0,Y 178.229,Z 407.166,A -85,B 0,C 180,E1 -25342.522,E2 -25342.522} C_VEL
LIN {X 0,Y 182.271,Z 395.248,A -85,B 0,C 180,E1 -25343.601,E2 -25343.601} C_VEL
LIN {X 0,Y 185.283,Z 383.275,A -85,B 0,C 180,E1 -25344.382,E2 -25344.382} C_VEL
LIN {X 0,Y 187.403,Z 370.292,A -85,B 0,C 180,E1 -25344.94,E2 -25344.94} C_VEL
LIN {X 0,Y 188.688,Z 356.325,A -85,B 0,C 180,E1 -25345.412,E2 -25345.412} C_VEL
LIN {X 0,Y 185.477,Z 348.007,A -85,B 0,C 180,E1 -25348.259,E2 -25348.259} C_VEL
LIN {X 0,Y 182.258,Z 340.679,A -85,B 0,C 180,E1 -25351.488,E2 -25351.488} C_VEL
LIN {X 0,Y 179.967,Z 335.938,A -85,B 0,C 180,E1 -25354.145,E2 -25354.145} C_VEL
LIN {X 0,Y 177.666,Z 331.528,A -85,B 0,C 180,E1 -25357.304,E2 -25357.304} C_VEL
LIN {X 0,Y 176.875,Z 330.265,A -85,B 0,C 180,E1 -25358.579,E2 -25358.579} C_VEL
LIN {X 0,Y 174.717,Z 326.283,A -85,B 0,C 180,E1 -25363.28,E2 -25363.28} C_VEL
LIN {X 0,Y 173.198,Z 324.517,A -85,B 0,C 180,E1 -25370.649,E2 -25370.649} C_VEL
LIN {X 0,Y 174.526,Z 325.628,A -85,B 0,C 180,E1 -25378.297,E2 -25378.297} C_VEL
LIN {X 0,Y 175.003,Z 326.292,A -85,B 0,C 180,E1 -25379.587,E2 -25379.587} C_VEL
LIN {X 0,Y 176.977,Z 329.982,A -85,B 0,C 180,E1 -25383.745,E2 -25383.745} C_VEL
LIN {X 0,Y 177.91,Z 331.587,A -85,B 0,C 180,E1 -25385.24,E2 -25385.24} C_VEL
LIN {X 0,Y 180.319,Z 335.651,A -85,B 0,C 180,E1 -25388.397,E2 -25388.397} C_VEL
LIN {X 0,Y 182.501,Z 339.448,A -85,B 0,C 180,E1 -25390.81,E2 -25390.81} C_VEL
LIN {X 0,Y 184.369,Z 343,A -85,B 0,C 180,E1 -25392.67,E2 -25392.67} C_VEL
LIN {X 0,Y 187.411,Z 349.955,A -85,B 0,C 180,E1 -25395.46,E2 -25395.46} C_VEL
LIN {X 0,Y 188.924,Z 353.772,A -85,B 0,C 180,E1 -25396.745,E2 -25396.745} C_VEL
LIN {X 0,Y 186.898,Z 373.049,A -85,B 0,C 180,E1 -25397.406,E2 -25397.406} C_VEL
LIN {X 0,Y 184.343,Z 385.868,A -85,B 0,C 180,E1 -25398.058,E2 -25398.058} C_VEL
LIN {X 0,Y 180.758,Z 398.385,A -85,B 0,C 180,E1 -25399.04,E2 -25399.04} C_VEL
LIN {X 0,Y 176.164,Z 410.535,A -85,B 0,C 180,E1 -25400.359,E2 -25400.359} C_VEL
LIN {X 0,Y 171.023,Z 421.464,A -85,B 0,C 180,E1 -25401.964,E2 -25401.964} C_VEL
LIN {X 0,Y 165.274,Z 431.47,A -85,B 0,C 180,E1 -25403.899,E2 -25403.899} C_VEL
LIN {X 0,Y 158.866,Z 440.984,A -85,B 0,C 180,E1 -25406.379,E2 -25406.379} C_VEL
LIN {X 0,Y 152.78,Z 448.768,A -85,B 0,C 180,E1 -25409.07,E2 -25409.07} C_VEL
LIN {X 0,Y 146.852,Z 455.357,A -85,B 0,C 180,E1 -25412.065,E2 -25412.065} C_VEL
LIN {X 0,Y 141.729,Z 460.4,A -85,B 0,C 180,E1 -25415.094,E2 -25415.094} C_VEL
LIN {X 0,Y 135.966,Z 465.418,A -85,B 0,C 180,E1 -25419.163,E2 -25419.163} C_VEL
LIN {X 0,Y 132.512,Z 468.061,A -85,B 0,C 180,E1 -25422.053,E2 -25422.053} C_VEL
LIN {X 0,Y 129.449,Z 470.167,A -85,B 0,C 180,E1 -25425.105,E2 -25425.105} C_VEL
LIN {X 0,Y 126.756,Z 471.815,A -85,B 0,C 180,E1 -25428.29,E2 -25428.29} C_VEL
LIN {X 0,Y 123.84,Z 473.209,A -85,B 0,C 180,E1 -25432.581,E2 -25432.581} C_VEL
LIN {X 0,Y 121.037,Z 473.928,A -85,B 0,C 180,E1 -25438.493,E2 -25438.493} C_VEL
LIN {X 0,Y 119.942,Z 473.738,A -85,B 0,C 180,E1 -25442.045,E2 -25442.045} C_VEL
LIN {X 0,Y 119.166,Z 473.092,A -85,B 0,C 180,E1 -25445.616,E2 -25445.616} C_VEL
LIN {X 0,Y 118.729,Z 471.216,A -85,B 0,C 180,E1 -25451.224,E2 -25451.224} C_VEL
LIN {X 0,Y 119.143,Z 467.373,A -85,B 0,C 180,E1 -25458.084,E2 -25458.084} C_VEL
LIN {X 0,Y 120.188,Z 462.819,A -85,B 0,C 180,E1 -25463.6,E2 -25463.6} C_VEL
LIN {X 0,Y 121.998,Z 456.65,A -85,B 0,C 180,E1 -25469.174,E2 -25469.174} C_VEL
LIN {X 0,Y 124.282,Z 449.606,A -85,B 0,C 180,E1 -25474.052,E2 -25474.052} C_VEL
LIN {X 0,Y 127.317,Z 440.75,A -85,B 0,C 180,E1 -25478.73,E2 -25478.73} C_VEL
LIN {X 0,Y 130.464,Z 431.647,A -85,B 0,C 180,E1 -25482.442,E2 -25482.442} C_VEL
LIN {X 0,Y 133.709,Z 421.62,A -85,B 0,C 180,E1 -25485.626,E2 -25485.626} C_VEL
LIN {X 0,Y 136.882,Z 410.479,A -85,B 0,C 180,E1 -25488.328,E2 -25488.328} C_VEL
LIN {X 0,Y 139.863,Z 397.986,A -85,B 0,C 180,E1 -25490.593,E2 -25490.593} C_VEL
LIN {X 0,Y 142.025,Z 386.167,A -85,B 0,C 180,E1 -25492.166,E2 -25492.166} C_VEL
LIN {X 0,Y 143.789,Z 373.408,A -85,B 0,C 180,E1 -25493.291,E2 -25493.291} C_VEL
LIN {X 0,Y 145.207,Z 354.84,A -85,B 0,C 180,E1 -25494.23,E2 -25494.23} C_VEL
LIN {X 0,Y 147.493,Z 319.365,A -85,B 0,C 180,E1 -25495.759,E2 -25495.759} C_VEL
LIN {X 0,Y 143.691,Z 308.273,A -85,B 0,C 180,E1 -25497.593,E2 -25497.593} C_VEL
LIN {X 0,Y 136.346,Z 294.301,A -85,B 0,C 180,E1 -25501.054,E2 -25501.054} C_VEL
LIN {X 0,Y 130.132,Z 284.425,A -85,B 0,C 180,E1 -25504.287,E2 -25504.287} C_VEL
LIN {X 0,Y 127.657,Z 280.779,A -85,B 0,C 180,E1 -25505.692,E2 -25505.692} C_VEL
LIN {X 0,Y 125.595,Z 277.809,A -85,B 0,C 180,E1 -25506.929,E2 -25506.929} C_VEL
LIN {X 0,Y 124.746,Z 276.636,A -85,B 0,C 180,E1 -25507.455,E2 -25507.455} C_VEL
LIN {X 0,Y 122.787,Z 274.369,A -85,B 0,C 180,E1 -25508.669,E2 -25508.669} C_VEL
LIN {X 0,Y 122.045,Z 272.281,A -85,B 0,C 180,E1 -25509.569,E2 -25509.569} C_VEL
LIN {X 0,Y 122.013,Z 271.818,A -85,B 0,C 180,E1 -25510.388,E2 -25510.388} C_VEL
LIN {X 0,Y 121.91,Z 271.799,A -85,B 0,C 180,E1 -25516.251,E2 -25516.251} C_VEL
LIN {X 0,Y 121.895,Z 271.756,A -85,B 0,C 180,E1 -25520.659,E2 -25520.659} C_VEL
LIN {X 0,Y 121.954,Z 271.774,A -85,B 0,C 180,E1 -25524.831,E2 -25524.831} C_VEL
LIN {X 0,Y 121.91,Z 271.755,A -85,B 0,C 180,E1 -25529.85,E2 -25529.85} C_VEL
LIN {X 0,Y 121.981,Z 271.766,A -85,B 0,C 180,E1 -25536.232,E2 -25536.232} C_VEL
LIN {X 0,Y 122.057,Z 271.769,A -85,B 0,C 180,E1 -25539.806,E2 -25539.806} C_VEL
LIN {X 0,Y 122.355,Z 271.693,A -85,B 0,C 180,E1 -25547.54,E2 -25547.54} C_VEL
LIN {X 0,Y 122.443,Z 271.725,A -85,B 0,C 180,E1 -25550.1,E2 -25550.1} C_VEL
LIN {X 0,Y 122.602,Z 271.648,A -85,B 0,C 180,E1 -25556.729,E2 -25556.729} C_VEL
LIN {X 0,Y 123.038,Z 271.603,A -85,B 0,C 180,E1 -25560.015,E2 -25560.015} C_VEL
